   STATUS[293].TimeStamp := 16#0000;
   STATUS[294].EXT.AlarmWarnUnAck := FALSE;
   STATUS[294].EXT.AckRequired := FALSE;
   STATUS[294].EXT.Maintanence := FALSE;
   STATUS[294].EXT.Operation := FALSE;
   STATUS[294].EXT.Forced := FALSE;
   STATUS[294].EXT.BIT29 := FALSE;
   STATUS[294].EXT.BIT30 := FALSE;
   STATUS[294].EXT.BIT31 := FALSE;
   STATUS[294].EXT.ModeBit1 := FALSE;
   STATUS[294].EXT.ModeBit2 := FALSE;
   STATUS[294].EXT.ModeBit3 := FALSE;
   STATUS[294].EXT.BIT19 := FALSE;
   STATUS[294].EXT.BIT20 := FALSE;
   STATUS[294].EXT.AlarmSuppressed := FALSE;
   STATUS[294].EXT.AlarmPresent := FALSE;
   STATUS[294].EXT.AlarmFailUnAck := FALSE;
   STATUS[294].Status := 0;
   STATUS[294].TimeStamp := 16#0000;
   STATUS[295].EXT.AlarmWarnUnAck := FALSE;
   STATUS[295].EXT.AckRequired := FALSE;
   STATUS[295].EXT.Maintanence := FALSE;
   STATUS[295].EXT.Operation := FALSE;
   STATUS[295].EXT.Forced := FALSE;
   STATUS[295].EXT.BIT29 := FALSE;
   STATUS[295].EXT.BIT30 := FALSE;
   STATUS[295].EXT.BIT31 := FALSE;
   STATUS[295].EXT.ModeBit1 := FALSE;
   STATUS[295].EXT.ModeBit2 := FALSE;
   STATUS[295].EXT.ModeBit3 := FALSE;
   STATUS[295].EXT.BIT19 := FALSE;
   STATUS[295].EXT.BIT20 := FALSE;
   STATUS[295].EXT.AlarmSuppressed := FALSE;
   STATUS[295].EXT.AlarmPresent := FALSE;
   STATUS[295].EXT.AlarmFailUnAck := FALSE;
   STATUS[295].Status := 0;
   STATUS[295].TimeStamp := 16#0000;
   STATUS[296].EXT.AlarmWarnUnAck := FALSE;
   STATUS[296].EXT.AckRequired := FALSE;
   STATUS[296].EXT.Maintanence := FALSE;
   STATUS[296].EXT.Operation := FALSE;
   STATUS[296].EXT.Forced := FALSE;
   STATUS[296].EXT.BIT29 := FALSE;
   STATUS[296].EXT.BIT30 := FALSE;
   STATUS[296].EXT.BIT31 := FALSE;
   STATUS[296].EXT.ModeBit1 := FALSE;
   STATUS[296].EXT.ModeBit2 := FALSE;
   STATUS[296].EXT.ModeBit3 := FALSE;
   STATUS[296].EXT.BIT19 := FALSE;
   STATUS[296].EXT.BIT20 := FALSE;
   STATUS[296].EXT.AlarmSuppressed := FALSE;
   STATUS[296].EXT.AlarmPresent := FALSE;
   STATUS[296].EXT.AlarmFailUnAck := FALSE;
   STATUS[296].Status := 0;
   STATUS[296].TimeStamp := 16#0000;
   STATUS[297].EXT.AlarmWarnUnAck := FALSE;
   STATUS[297].EXT.AckRequired := FALSE;
   STATUS[297].EXT.Maintanence := FALSE;
   STATUS[297].EXT.Operation := FALSE;
   STATUS[297].EXT.Forced := FALSE;
   STATUS[297].EXT.BIT29 := FALSE;
   STATUS[297].EXT.BIT30 := FALSE;
   STATUS[297].EXT.BIT31 := FALSE;
   STATUS[297].EXT.ModeBit1 := FALSE;
   STATUS[297].EXT.ModeBit2 := FALSE;
   STATUS[297].EXT.ModeBit3 := FALSE;
   STATUS[297].EXT.BIT19 := FALSE;
   STATUS[297].EXT.BIT20 := FALSE;
   STATUS[297].EXT.AlarmSuppressed := FALSE;
   STATUS[297].EXT.AlarmPresent := FALSE;
   STATUS[297].EXT.AlarmFailUnAck := FALSE;
   STATUS[297].Status := 0;
   STATUS[297].TimeStamp := 16#0000;
   STATUS[298].EXT.AlarmWarnUnAck := FALSE;
   STATUS[298].EXT.AckRequired := FALSE;
   STATUS[298].EXT.Maintanence := FALSE;
   STATUS[298].EXT.Operation := FALSE;
   STATUS[298].EXT.Forced := FALSE;
   STATUS[298].EXT.BIT29 := FALSE;
   STATUS[298].EXT.BIT30 := FALSE;
   STATUS[298].EXT.BIT31 := FALSE;
   STATUS[298].EXT.ModeBit1 := FALSE;
   STATUS[298].EXT.ModeBit2 := FALSE;
   STATUS[298].EXT.ModeBit3 := FALSE;
   STATUS[298].EXT.BIT19 := FALSE;
   STATUS[298].EXT.BIT20 := FALSE;
   STATUS[298].EXT.AlarmSuppressed := FALSE;
   STATUS[298].EXT.AlarmPresent := FALSE;
   STATUS[298].EXT.AlarmFailUnAck := FALSE;
   STATUS[298].Status := 0;
   STATUS[298].TimeStamp := 16#0000;
   STATUS[299].EXT.AlarmWarnUnAck := FALSE;
   STATUS[299].EXT.AckRequired := FALSE;
   STATUS[299].EXT.Maintanence := FALSE;
   STATUS[299].EXT.Operation := FALSE;
   STATUS[299].EXT.Forced := FALSE;
   STATUS[299].EXT.BIT29 := FALSE;
   STATUS[299].EXT.BIT30 := FALSE;
   STATUS[299].EXT.BIT31 := FALSE;
   STATUS[299].EXT.ModeBit1 := FALSE;
   STATUS[299].EXT.ModeBit2 := FALSE;
   STATUS[299].EXT.ModeBit3 := FALSE;
   STATUS[299].EXT.BIT19 := FALSE;
   STATUS[299].EXT.BIT20 := FALSE;
   STATUS[299].EXT.AlarmSuppressed := FALSE;
   STATUS[299].EXT.AlarmPresent := FALSE;
   STATUS[299].EXT.AlarmFailUnAck := FALSE;
   STATUS[299].Status := 0;
   STATUS[299].TimeStamp := 16#0000;
   STATUS[300].EXT.AlarmWarnUnAck := FALSE;
   STATUS[300].EXT.AckRequired := FALSE;
   STATUS[300].EXT.Maintanence := FALSE;
   STATUS[300].EXT.Operation := FALSE;
   STATUS[300].EXT.Forced := FALSE;
   STATUS[300].EXT.BIT29 := FALSE;
   STATUS[300].EXT.BIT30 := FALSE;
   STATUS[300].EXT.BIT31 := FALSE;
   STATUS[300].EXT.ModeBit1 := FALSE;
   STATUS[300].EXT.ModeBit2 := FALSE;
   STATUS[300].EXT.ModeBit3 := FALSE;
   STATUS[300].EXT.BIT19 := FALSE;
   STATUS[300].EXT.BIT20 := FALSE;
   STATUS[300].EXT.AlarmSuppressed := FALSE;
   STATUS[300].EXT.AlarmPresent := FALSE;
   STATUS[300].EXT.AlarmFailUnAck := FALSE;
   STATUS[300].Status := 0;
   STATUS[300].TimeStamp := 16#0000;
   STATUS[301].EXT.AlarmWarnUnAck := FALSE;
   STATUS[301].EXT.AckRequired := FALSE;
   STATUS[301].EXT.Maintanence := FALSE;
   STATUS[301].EXT.Operation := FALSE;
   STATUS[301].EXT.Forced := FALSE;
   STATUS[301].EXT.BIT29 := FALSE;
   STATUS[301].EXT.BIT30 := FALSE;
   STATUS[301].EXT.BIT31 := FALSE;
   STATUS[301].EXT.ModeBit1 := FALSE;
   STATUS[301].EXT.ModeBit2 := FALSE;
   STATUS[301].EXT.ModeBit3 := FALSE;
   STATUS[301].EXT.BIT19 := FALSE;
   STATUS[301].EXT.BIT20 := FALSE;
   STATUS[301].EXT.AlarmSuppressed := FALSE;
   STATUS[301].EXT.AlarmPresent := FALSE;
   STATUS[301].EXT.AlarmFailUnAck := FALSE;
   STATUS[301].Status := 0;
   STATUS[301].TimeStamp := 16#0000;
   STATUS[302].EXT.AlarmWarnUnAck := FALSE;
   STATUS[302].EXT.AckRequired := FALSE;
   STATUS[302].EXT.Maintanence := FALSE;
   STATUS[302].EXT.Operation := FALSE;
   STATUS[302].EXT.Forced := FALSE;
   STATUS[302].EXT.BIT29 := FALSE;
   STATUS[302].EXT.BIT30 := FALSE;
   STATUS[302].EXT.BIT31 := FALSE;
   STATUS[302].EXT.ModeBit1 := FALSE;
   STATUS[302].EXT.ModeBit2 := FALSE;
   STATUS[302].EXT.ModeBit3 := FALSE;
   STATUS[302].EXT.BIT19 := FALSE;
   STATUS[302].EXT.BIT20 := FALSE;
   STATUS[302].EXT.AlarmSuppressed := FALSE;
   STATUS[302].EXT.AlarmPresent := FALSE;
   STATUS[302].EXT.AlarmFailUnAck := FALSE;
   STATUS[302].Status := 0;
   STATUS[302].TimeStamp := 16#0000;
   STATUS[303].EXT.AlarmWarnUnAck := FALSE;
   STATUS[303].EXT.AckRequired := FALSE;
   STATUS[303].EXT.Maintanence := FALSE;
   STATUS[303].EXT.Operation := FALSE;
   STATUS[303].EXT.Forced := FALSE;
   STATUS[303].EXT.BIT29 := FALSE;
   STATUS[303].EXT.BIT30 := FALSE;
   STATUS[303].EXT.BIT31 := FALSE;
   STATUS[303].EXT.ModeBit1 := FALSE;
   STATUS[303].EXT.ModeBit2 := FALSE;
   STATUS[303].EXT.ModeBit3 := FALSE;
   STATUS[303].EXT.BIT19 := FALSE;
   STATUS[303].EXT.BIT20 := FALSE;
   STATUS[303].EXT.AlarmSuppressed := FALSE;
   STATUS[303].EXT.AlarmPresent := FALSE;
   STATUS[303].EXT.AlarmFailUnAck := FALSE;
   STATUS[303].Status := 0;
   STATUS[303].TimeStamp := 16#0000;
   STATUS[304].EXT.AlarmWarnUnAck := FALSE;
   STATUS[304].EXT.AckRequired := FALSE;
   STATUS[304].EXT.Maintanence := FALSE;
   STATUS[304].EXT.Operation := FALSE;
   STATUS[304].EXT.Forced := FALSE;
   STATUS[304].EXT.BIT29 := FALSE;
   STATUS[304].EXT.BIT30 := FALSE;
   STATUS[304].EXT.BIT31 := FALSE;
   STATUS[304].EXT.ModeBit1 := FALSE;
   STATUS[304].EXT.ModeBit2 := FALSE;
   STATUS[304].EXT.ModeBit3 := FALSE;
   STATUS[304].EXT.BIT19 := FALSE;
   STATUS[304].EXT.BIT20 := FALSE;
   STATUS[304].EXT.AlarmSuppressed := FALSE;
   STATUS[304].EXT.AlarmPresent := FALSE;
   STATUS[304].EXT.AlarmFailUnAck := FALSE;
   STATUS[304].Status := 0;
   STATUS[304].TimeStamp := 16#0000;
   STATUS[305].EXT.AlarmWarnUnAck := FALSE;
   STATUS[305].EXT.AckRequired := FALSE;
   STATUS[305].EXT.Maintanence := FALSE;
   STATUS[305].EXT.Operation := FALSE;
   STATUS[305].EXT.Forced := FALSE;
   STATUS[305].EXT.BIT29 := FALSE;
   STATUS[305].EXT.BIT30 := FALSE;
   STATUS[305].EXT.BIT31 := FALSE;
   STATUS[305].EXT.ModeBit1 := FALSE;
   STATUS[305].EXT.ModeBit2 := FALSE;
   STATUS[305].EXT.ModeBit3 := FALSE;
   STATUS[305].EXT.BIT19 := FALSE;
   STATUS[305].EXT.BIT20 := FALSE;
   STATUS[305].EXT.AlarmSuppressed := FALSE;
   STATUS[305].EXT.AlarmPresent := FALSE;
   STATUS[305].EXT.AlarmFailUnAck := FALSE;
   STATUS[305].Status := 0;
   STATUS[305].TimeStamp := 16#0000;
   STATUS[306].EXT.AlarmWarnUnAck := FALSE;
   STATUS[306].EXT.AckRequired := FALSE;
   STATUS[306].EXT.Maintanence := FALSE;
   STATUS[306].EXT.Operation := FALSE;
   STATUS[306].EXT.Forced := FALSE;
   STATUS[306].EXT.BIT29 := FALSE;
   STATUS[306].EXT.BIT30 := FALSE;
   STATUS[306].EXT.BIT31 := FALSE;
   STATUS[306].EXT.ModeBit1 := FALSE;
   STATUS[306].EXT.ModeBit2 := FALSE;
   STATUS[306].EXT.ModeBit3 := FALSE;
   STATUS[306].EXT.BIT19 := FALSE;
   STATUS[306].EXT.BIT20 := FALSE;
   STATUS[306].EXT.AlarmSuppressed := FALSE;
   STATUS[306].EXT.AlarmPresent := FALSE;
   STATUS[306].EXT.AlarmFailUnAck := FALSE;
   STATUS[306].Status := 0;
   STATUS[306].TimeStamp := 16#0000;
   STATUS[307].EXT.AlarmWarnUnAck := FALSE;
   STATUS[307].EXT.AckRequired := FALSE;
   STATUS[307].EXT.Maintanence := FALSE;
   STATUS[307].EXT.Operation := FALSE;
   STATUS[307].EXT.Forced := FALSE;
   STATUS[307].EXT.BIT29 := FALSE;
   STATUS[307].EXT.BIT30 := FALSE;
   STATUS[307].EXT.BIT31 := FALSE;
   STATUS[307].EXT.ModeBit1 := FALSE;
   STATUS[307].EXT.ModeBit2 := FALSE;
   STATUS[307].EXT.ModeBit3 := FALSE;
   STATUS[307].EXT.BIT19 := FALSE;
   STATUS[307].EXT.BIT20 := FALSE;
   STATUS[307].EXT.AlarmSuppressed := FALSE;
   STATUS[307].EXT.AlarmPresent := FALSE;
   STATUS[307].EXT.AlarmFailUnAck := FALSE;
   STATUS[307].Status := 0;
   STATUS[307].TimeStamp := 16#0000;
   STATUS[308].EXT.AlarmWarnUnAck := FALSE;
   STATUS[308].EXT.AckRequired := FALSE;
   STATUS[308].EXT.Maintanence := FALSE;
   STATUS[308].EXT.Operation := FALSE;
   STATUS[308].EXT.Forced := FALSE;
   STATUS[308].EXT.BIT29 := FALSE;
   STATUS[308].EXT.BIT30 := FALSE;
   STATUS[308].EXT.BIT31 := FALSE;
   STATUS[308].EXT.ModeBit1 := FALSE;
   STATUS[308].EXT.ModeBit2 := FALSE;
   STATUS[308].EXT.ModeBit3 := FALSE;
   STATUS[308].EXT.BIT19 := FALSE;
   STATUS[308].EXT.BIT20 := FALSE;
   STATUS[308].EXT.AlarmSuppressed := FALSE;
   STATUS[308].EXT.AlarmPresent := FALSE;
   STATUS[308].EXT.AlarmFailUnAck := FALSE;
   STATUS[308].Status := 0;
   STATUS[308].TimeStamp := 16#0000;
   STATUS[309].EXT.AlarmWarnUnAck := FALSE;
   STATUS[309].EXT.AckRequired := FALSE;
   STATUS[309].EXT.Maintanence := FALSE;
   STATUS[309].EXT.Operation := FALSE;
   STATUS[309].EXT.Forced := FALSE;
   STATUS[309].EXT.BIT29 := FALSE;
   STATUS[309].EXT.BIT30 := FALSE;
   STATUS[309].EXT.BIT31 := FALSE;
   STATUS[309].EXT.ModeBit1 := FALSE;
   STATUS[309].EXT.ModeBit2 := FALSE;
   STATUS[309].EXT.ModeBit3 := FALSE;
   STATUS[309].EXT.BIT19 := FALSE;
   STATUS[309].EXT.BIT20 := FALSE;
   STATUS[309].EXT.AlarmSuppressed := FALSE;
   STATUS[309].EXT.AlarmPresent := FALSE;
   STATUS[309].EXT.AlarmFailUnAck := FALSE;
   STATUS[309].Status := 0;
   STATUS[309].TimeStamp := 16#0000;
   STATUS[310].EXT.AlarmWarnUnAck := FALSE;
   STATUS[310].EXT.AckRequired := FALSE;
   STATUS[310].EXT.Maintanence := FALSE;
   STATUS[310].EXT.Operation := FALSE;
   STATUS[310].EXT.Forced := FALSE;
   STATUS[310].EXT.BIT29 := FALSE;
   STATUS[310].EXT.BIT30 := FALSE;
   STATUS[310].EXT.BIT31 := FALSE;
   STATUS[310].EXT.ModeBit1 := FALSE;
   STATUS[310].EXT.ModeBit2 := FALSE;
   STATUS[310].EXT.ModeBit3 := FALSE;
   STATUS[310].EXT.BIT19 := FALSE;
   STATUS[310].EXT.BIT20 := FALSE;
   STATUS[310].EXT.AlarmSuppressed := FALSE;
   STATUS[310].EXT.AlarmPresent := FALSE;
   STATUS[310].EXT.AlarmFailUnAck := FALSE;
   STATUS[310].Status := 0;
   STATUS[310].TimeStamp := 16#0000;
   STATUS[311].EXT.AlarmWarnUnAck := FALSE;
   STATUS[311].EXT.AckRequired := FALSE;
   STATUS[311].EXT.Maintanence := FALSE;
   STATUS[311].EXT.Operation := FALSE;
   STATUS[311].EXT.Forced := FALSE;
   STATUS[311].EXT.BIT29 := FALSE;
   STATUS[311].EXT.BIT30 := FALSE;
   STATUS[311].EXT.BIT31 := FALSE;
   STATUS[311].EXT.ModeBit1 := FALSE;
   STATUS[311].EXT.ModeBit2 := FALSE;
   STATUS[311].EXT.ModeBit3 := FALSE;
   STATUS[311].EXT.BIT19 := FALSE;
   STATUS[311].EXT.BIT20 := FALSE;
   STATUS[311].EXT.AlarmSuppressed := FALSE;
   STATUS[311].EXT.AlarmPresent := FALSE;
   STATUS[311].EXT.AlarmFailUnAck := FALSE;
   STATUS[311].Status := 0;
   STATUS[311].TimeStamp := 16#0000;
   STATUS[312].EXT.AlarmWarnUnAck := FALSE;
   STATUS[312].EXT.AckRequired := FALSE;
   STATUS[312].EXT.Maintanence := FALSE;
   STATUS[312].EXT.Operation := FALSE;
   STATUS[312].EXT.Forced := FALSE;
   STATUS[312].EXT.BIT29 := FALSE;
   STATUS[312].EXT.BIT30 := FALSE;
   STATUS[312].EXT.BIT31 := FALSE;
   STATUS[312].EXT.ModeBit1 := FALSE;
   STATUS[312].EXT.ModeBit2 := FALSE;
   STATUS[312].EXT.ModeBit3 := FALSE;
   STATUS[312].EXT.BIT19 := FALSE;
   STATUS[312].EXT.BIT20 := FALSE;
   STATUS[312].EXT.AlarmSuppressed := FALSE;
   STATUS[312].EXT.AlarmPresent := FALSE;
   STATUS[312].EXT.AlarmFailUnAck := FALSE;
   STATUS[312].Status := 0;
   STATUS[312].TimeStamp := 16#0000;
   STATUS[313].EXT.AlarmWarnUnAck := FALSE;
   STATUS[313].EXT.AckRequired := FALSE;
   STATUS[313].EXT.Maintanence := FALSE;
   STATUS[313].EXT.Operation := FALSE;
   STATUS[313].EXT.Forced := FALSE;
   STATUS[313].EXT.BIT29 := FALSE;
   STATUS[313].EXT.BIT30 := FALSE;
   STATUS[313].EXT.BIT31 := FALSE;
   STATUS[313].EXT.ModeBit1 := FALSE;
   STATUS[313].EXT.ModeBit2 := FALSE;
   STATUS[313].EXT.ModeBit3 := FALSE;
   STATUS[313].EXT.BIT19 := FALSE;
   STATUS[313].EXT.BIT20 := FALSE;
   STATUS[313].EXT.AlarmSuppressed := FALSE;
   STATUS[313].EXT.AlarmPresent := FALSE;
   STATUS[313].EXT.AlarmFailUnAck := FALSE;
   STATUS[313].Status := 0;
   STATUS[313].TimeStamp := 16#0000;
   STATUS[314].EXT.AlarmWarnUnAck := FALSE;
   STATUS[314].EXT.AckRequired := FALSE;
   STATUS[314].EXT.Maintanence := FALSE;
   STATUS[314].EXT.Operation := FALSE;
   STATUS[314].EXT.Forced := FALSE;
   STATUS[314].EXT.BIT29 := FALSE;
   STATUS[314].EXT.BIT30 := FALSE;
   STATUS[314].EXT.BIT31 := FALSE;
   STATUS[314].EXT.ModeBit1 := FALSE;
   STATUS[314].EXT.ModeBit2 := FALSE;
   STATUS[314].EXT.ModeBit3 := FALSE;
   STATUS[314].EXT.BIT19 := FALSE;
   STATUS[314].EXT.BIT20 := FALSE;
   STATUS[314].EXT.AlarmSuppressed := FALSE;
   STATUS[314].EXT.AlarmPresent := FALSE;
   STATUS[314].EXT.AlarmFailUnAck := FALSE;
   STATUS[314].Status := 0;
   STATUS[314].TimeStamp := 16#0000;
   STATUS[315].EXT.AlarmWarnUnAck := FALSE;
   STATUS[315].EXT.AckRequired := FALSE;
   STATUS[315].EXT.Maintanence := FALSE;
   STATUS[315].EXT.Operation := FALSE;
   STATUS[315].EXT.Forced := FALSE;
   STATUS[315].EXT.BIT29 := FALSE;
   STATUS[315].EXT.BIT30 := FALSE;
   STATUS[315].EXT.BIT31 := FALSE;
   STATUS[315].EXT.ModeBit1 := FALSE;
   STATUS[315].EXT.ModeBit2 := FALSE;
   STATUS[315].EXT.ModeBit3 := FALSE;
   STATUS[315].EXT.BIT19 := FALSE;
   STATUS[315].EXT.BIT20 := FALSE;
   STATUS[315].EXT.AlarmSuppressed := FALSE;
   STATUS[315].EXT.AlarmPresent := FALSE;
   STATUS[315].EXT.AlarmFailUnAck := FALSE;
   STATUS[315].Status := 0;
   STATUS[315].TimeStamp := 16#0000;
   STATUS[316].EXT.AlarmWarnUnAck := FALSE;
   STATUS[316].EXT.AckRequired := FALSE;
   STATUS[316].EXT.Maintanence := FALSE;
   STATUS[316].EXT.Operation := FALSE;
   STATUS[316].EXT.Forced := FALSE;
   STATUS[316].EXT.BIT29 := FALSE;
   STATUS[316].EXT.BIT30 := FALSE;
   STATUS[316].EXT.BIT31 := FALSE;
   STATUS[316].EXT.ModeBit1 := FALSE;
   STATUS[316].EXT.ModeBit2 := FALSE;
   STATUS[316].EXT.ModeBit3 := FALSE;
   STATUS[316].EXT.BIT19 := FALSE;
   STATUS[316].EXT.BIT20 := FALSE;
   STATUS[316].EXT.AlarmSuppressed := FALSE;
   STATUS[316].EXT.AlarmPresent := FALSE;
   STATUS[316].EXT.AlarmFailUnAck := FALSE;
   STATUS[316].Status := 0;
   STATUS[316].TimeStamp := 16#0000;
   STATUS[317].EXT.AlarmWarnUnAck := FALSE;
   STATUS[317].EXT.AckRequired := FALSE;
   STATUS[317].EXT.Maintanence := FALSE;
   STATUS[317].EXT.Operation := FALSE;
   STATUS[317].EXT.Forced := FALSE;
   STATUS[317].EXT.BIT29 := FALSE;
   STATUS[317].EXT.BIT30 := FALSE;
   STATUS[317].EXT.BIT31 := FALSE;
   STATUS[317].EXT.ModeBit1 := FALSE;
   STATUS[317].EXT.ModeBit2 := FALSE;
   STATUS[317].EXT.ModeBit3 := FALSE;
   STATUS[317].EXT.BIT19 := FALSE;
   STATUS[317].EXT.BIT20 := FALSE;
   STATUS[317].EXT.AlarmSuppressed := FALSE;
   STATUS[317].EXT.AlarmPresent := FALSE;
   STATUS[317].EXT.AlarmFailUnAck := FALSE;
   STATUS[317].Status := 0;
   STATUS[317].TimeStamp := 16#0000;
   STATUS[318].EXT.AlarmWarnUnAck := FALSE;
   STATUS[318].EXT.AckRequired := FALSE;
   STATUS[318].EXT.Maintanence := FALSE;
   STATUS[318].EXT.Operation := FALSE;
   STATUS[318].EXT.Forced := FALSE;
   STATUS[318].EXT.BIT29 := FALSE;
   STATUS[318].EXT.BIT30 := FALSE;
   STATUS[318].EXT.BIT31 := FALSE;
   STATUS[318].EXT.ModeBit1 := FALSE;
   STATUS[318].EXT.ModeBit2 := FALSE;
   STATUS[318].EXT.ModeBit3 := FALSE;
   STATUS[318].EXT.BIT19 := FALSE;
   STATUS[318].EXT.BIT20 := FALSE;
   STATUS[318].EXT.AlarmSuppressed := FALSE;
   STATUS[318].EXT.AlarmPresent := FALSE;
   STATUS[318].EXT.AlarmFailUnAck := FALSE;
   STATUS[318].Status := 0;
   STATUS[318].TimeStamp := 16#0000;
   STATUS[319].EXT.AlarmWarnUnAck := FALSE;
   STATUS[319].EXT.AckRequired := FALSE;
   STATUS[319].EXT.Maintanence := FALSE;
   STATUS[319].EXT.Operation := FALSE;
   STATUS[319].EXT.Forced := FALSE;
   STATUS[319].EXT.BIT29 := FALSE;
   STATUS[319].EXT.BIT30 := FALSE;
   STATUS[319].EXT.BIT31 := FALSE;
   STATUS[319].EXT.ModeBit1 := FALSE;
   STATUS[319].EXT.ModeBit2 := FALSE;
   STATUS[319].EXT.ModeBit3 := FALSE;
   STATUS[319].EXT.BIT19 := FALSE;
   STATUS[319].EXT.BIT20 := FALSE;
   STATUS[319].EXT.AlarmSuppressed := FALSE;
   STATUS[319].EXT.AlarmPresent := FALSE;
   STATUS[319].EXT.AlarmFailUnAck := FALSE;
   STATUS[319].Status := 0;
   STATUS[319].TimeStamp := 16#0000;
   STATUS[320].EXT.AlarmWarnUnAck := FALSE;
   STATUS[320].EXT.AckRequired := FALSE;
   STATUS[320].EXT.Maintanence := FALSE;
   STATUS[320].EXT.Operation := FALSE;
   STATUS[320].EXT.Forced := FALSE;
   STATUS[320].EXT.BIT29 := FALSE;
   STATUS[320].EXT.BIT30 := FALSE;
   STATUS[320].EXT.BIT31 := FALSE;
   STATUS[320].EXT.ModeBit1 := FALSE;
   STATUS[320].EXT.ModeBit2 := FALSE;
   STATUS[320].EXT.ModeBit3 := FALSE;
   STATUS[320].EXT.BIT19 := FALSE;
   STATUS[320].EXT.BIT20 := FALSE;
   STATUS[320].EXT.AlarmSuppressed := FALSE;
   STATUS[320].EXT.AlarmPresent := FALSE;
   STATUS[320].EXT.AlarmFailUnAck := FALSE;
   STATUS[320].Status := 0;
   STATUS[320].TimeStamp := 16#0000;
   STATUS[321].EXT.AlarmWarnUnAck := FALSE;
   STATUS[321].EXT.AckRequired := FALSE;
   STATUS[321].EXT.Maintanence := FALSE;
   STATUS[321].EXT.Operation := FALSE;
   STATUS[321].EXT.Forced := FALSE;
   STATUS[321].EXT.BIT29 := FALSE;
   STATUS[321].EXT.BIT30 := FALSE;
   STATUS[321].EXT.BIT31 := FALSE;
   STATUS[321].EXT.ModeBit1 := FALSE;
   STATUS[321].EXT.ModeBit2 := FALSE;
   STATUS[321].EXT.ModeBit3 := FALSE;
   STATUS[321].EXT.BIT19 := FALSE;
   STATUS[321].EXT.BIT20 := FALSE;
   STATUS[321].EXT.AlarmSuppressed := FALSE;
   STATUS[321].EXT.AlarmPresent := FALSE;
   STATUS[321].EXT.AlarmFailUnAck := FALSE;
   STATUS[321].Status := 0;
   STATUS[321].TimeStamp := 16#0000;
   STATUS[322].EXT.AlarmWarnUnAck := FALSE;
   STATUS[322].EXT.AckRequired := FALSE;
   STATUS[322].EXT.Maintanence := FALSE;
   STATUS[322].EXT.Operation := FALSE;
   STATUS[322].EXT.Forced := FALSE;
   STATUS[322].EXT.BIT29 := FALSE;
   STATUS[322].EXT.BIT30 := FALSE;
   STATUS[322].EXT.BIT31 := FALSE;
   STATUS[322].EXT.ModeBit1 := FALSE;
   STATUS[322].EXT.ModeBit2 := FALSE;
   STATUS[322].EXT.ModeBit3 := FALSE;
   STATUS[322].EXT.BIT19 := FALSE;
   STATUS[322].EXT.BIT20 := FALSE;
   STATUS[322].EXT.AlarmSuppressed := FALSE;
   STATUS[322].EXT.AlarmPresent := FALSE;
   STATUS[322].EXT.AlarmFailUnAck := FALSE;
   STATUS[322].Status := 0;
   STATUS[322].TimeStamp := 16#0000;
   STATUS[323].EXT.AlarmWarnUnAck := FALSE;
   STATUS[323].EXT.AckRequired := FALSE;
   STATUS[323].EXT.Maintanence := FALSE;
   STATUS[323].EXT.Operation := FALSE;
   STATUS[323].EXT.Forced := FALSE;
   STATUS[323].EXT.BIT29 := FALSE;
   STATUS[323].EXT.BIT30 := FALSE;
   STATUS[323].EXT.BIT31 := FALSE;
   STATUS[323].EXT.ModeBit1 := FALSE;
   STATUS[323].EXT.ModeBit2 := FALSE;
   STATUS[323].EXT.ModeBit3 := FALSE;
   STATUS[323].EXT.BIT19 := FALSE;
   STATUS[323].EXT.BIT20 := FALSE;
   STATUS[323].EXT.AlarmSuppressed := FALSE;
   STATUS[323].EXT.AlarmPresent := FALSE;
   STATUS[323].EXT.AlarmFailUnAck := FALSE;
   STATUS[323].Status := 0;
   STATUS[323].TimeStamp := 16#0000;
   STATUS[324].EXT.AlarmWarnUnAck := FALSE;
   STATUS[324].EXT.AckRequired := FALSE;
   STATUS[324].EXT.Maintanence := FALSE;
   STATUS[324].EXT.Operation := FALSE;
   STATUS[324].EXT.Forced := FALSE;
   STATUS[324].EXT.BIT29 := FALSE;
   STATUS[324].EXT.BIT30 := FALSE;
   STATUS[324].EXT.BIT31 := FALSE;
   STATUS[324].EXT.ModeBit1 := FALSE;
   STATUS[324].EXT.ModeBit2 := FALSE;
   STATUS[324].EXT.ModeBit3 := FALSE;
   STATUS[324].EXT.BIT19 := FALSE;
   STATUS[324].EXT.BIT20 := FALSE;
   STATUS[324].EXT.AlarmSuppressed := FALSE;
   STATUS[324].EXT.AlarmPresent := FALSE;
   STATUS[324].EXT.AlarmFailUnAck := FALSE;
   STATUS[324].Status := 0;
   STATUS[324].TimeStamp := 16#0000;
   STATUS[325].EXT.AlarmWarnUnAck := FALSE;
   STATUS[325].EXT.AckRequired := FALSE;
   STATUS[325].EXT.Maintanence := FALSE;
   STATUS[325].EXT.Operation := FALSE;
   STATUS[325].EXT.Forced := FALSE;
   STATUS[325].EXT.BIT29 := FALSE;
   STATUS[325].EXT.BIT30 := FALSE;
   STATUS[325].EXT.BIT31 := FALSE;
   STATUS[325].EXT.ModeBit1 := FALSE;
   STATUS[325].EXT.ModeBit2 := FALSE;
   STATUS[325].EXT.ModeBit3 := FALSE;
   STATUS[325].EXT.BIT19 := FALSE;
   STATUS[325].EXT.BIT20 := FALSE;
   STATUS[325].EXT.AlarmSuppressed := FALSE;
   STATUS[325].EXT.AlarmPresent := FALSE;
   STATUS[325].EXT.AlarmFailUnAck := FALSE;
   STATUS[325].Status := 0;
   STATUS[325].TimeStamp := 16#0000;
   STATUS[326].EXT.AlarmWarnUnAck := FALSE;
   STATUS[326].EXT.AckRequired := FALSE;
   STATUS[326].EXT.Maintanence := FALSE;
   STATUS[326].EXT.Operation := FALSE;
   STATUS[326].EXT.Forced := FALSE;
   STATUS[326].EXT.BIT29 := FALSE;
   STATUS[326].EXT.BIT30 := FALSE;
   STATUS[326].EXT.BIT31 := FALSE;
   STATUS[326].EXT.ModeBit1 := FALSE;
   STATUS[326].EXT.ModeBit2 := FALSE;
   STATUS[326].EXT.ModeBit3 := FALSE;
   STATUS[326].EXT.BIT19 := FALSE;
   STATUS[326].EXT.BIT20 := FALSE;
   STATUS[326].EXT.AlarmSuppressed := FALSE;
   STATUS[326].EXT.AlarmPresent := FALSE;
   STATUS[326].EXT.AlarmFailUnAck := FALSE;
   STATUS[326].Status := 0;
   STATUS[326].TimeStamp := 16#0000;
   STATUS[327].EXT.AlarmWarnUnAck := FALSE;
   STATUS[327].EXT.AckRequired := FALSE;
   STATUS[327].EXT.Maintanence := FALSE;
   STATUS[327].EXT.Operation := FALSE;
   STATUS[327].EXT.Forced := FALSE;
   STATUS[327].EXT.BIT29 := FALSE;
   STATUS[327].EXT.BIT30 := FALSE;
   STATUS[327].EXT.BIT31 := FALSE;
   STATUS[327].EXT.ModeBit1 := FALSE;
   STATUS[327].EXT.ModeBit2 := FALSE;
   STATUS[327].EXT.ModeBit3 := FALSE;
   STATUS[327].EXT.BIT19 := FALSE;
   STATUS[327].EXT.BIT20 := FALSE;
   STATUS[327].EXT.AlarmSuppressed := FALSE;
   STATUS[327].EXT.AlarmPresent := FALSE;
   STATUS[327].EXT.AlarmFailUnAck := FALSE;
   STATUS[327].Status := 0;
   STATUS[327].TimeStamp := 16#0000;
   STATUS[328].EXT.AlarmWarnUnAck := FALSE;
   STATUS[328].EXT.AckRequired := FALSE;
   STATUS[328].EXT.Maintanence := FALSE;
   STATUS[328].EXT.Operation := FALSE;
   STATUS[328].EXT.Forced := FALSE;
   STATUS[328].EXT.BIT29 := FALSE;
   STATUS[328].EXT.BIT30 := FALSE;
   STATUS[328].EXT.BIT31 := FALSE;
   STATUS[328].EXT.ModeBit1 := FALSE;
   STATUS[328].EXT.ModeBit2 := FALSE;
   STATUS[328].EXT.ModeBit3 := FALSE;
   STATUS[328].EXT.BIT19 := FALSE;
   STATUS[328].EXT.BIT20 := FALSE;
   STATUS[328].EXT.AlarmSuppressed := FALSE;
   STATUS[328].EXT.AlarmPresent := FALSE;
   STATUS[328].EXT.AlarmFailUnAck := FALSE;
   STATUS[328].Status := 0;
   STATUS[328].TimeStamp := 16#0000;
   STATUS[329].EXT.AlarmWarnUnAck := FALSE;
   STATUS[329].EXT.AckRequired := FALSE;
   STATUS[329].EXT.Maintanence := FALSE;
   STATUS[329].EXT.Operation := FALSE;
   STATUS[329].EXT.Forced := FALSE;
   STATUS[329].EXT.BIT29 := FALSE;
   STATUS[329].EXT.BIT30 := FALSE;
   STATUS[329].EXT.BIT31 := FALSE;
   STATUS[329].EXT.ModeBit1 := FALSE;
   STATUS[329].EXT.ModeBit2 := FALSE;
   STATUS[329].EXT.ModeBit3 := FALSE;
   STATUS[329].EXT.BIT19 := FALSE;
   STATUS[329].EXT.BIT20 := FALSE;
   STATUS[329].EXT.AlarmSuppressed := FALSE;
   STATUS[329].EXT.AlarmPresent := FALSE;
   STATUS[329].EXT.AlarmFailUnAck := FALSE;
   STATUS[329].Status := 0;
   STATUS[329].TimeStamp := 16#0000;
   STATUS[330].EXT.AlarmWarnUnAck := FALSE;
   STATUS[330].EXT.AckRequired := FALSE;
   STATUS[330].EXT.Maintanence := FALSE;
   STATUS[330].EXT.Operation := FALSE;
   STATUS[330].EXT.Forced := FALSE;
   STATUS[330].EXT.BIT29 := FALSE;
   STATUS[330].EXT.BIT30 := FALSE;
   STATUS[330].EXT.BIT31 := FALSE;
   STATUS[330].EXT.ModeBit1 := FALSE;
   STATUS[330].EXT.ModeBit2 := FALSE;
   STATUS[330].EXT.ModeBit3 := FALSE;
   STATUS[330].EXT.BIT19 := FALSE;
   STATUS[330].EXT.BIT20 := FALSE;
   STATUS[330].EXT.AlarmSuppressed := FALSE;
   STATUS[330].EXT.AlarmPresent := FALSE;
   STATUS[330].EXT.AlarmFailUnAck := FALSE;
   STATUS[330].Status := 0;
   STATUS[330].TimeStamp := 16#0000;
   STATUS[331].EXT.AlarmWarnUnAck := FALSE;
   STATUS[331].EXT.AckRequired := FALSE;
   STATUS[331].EXT.Maintanence := FALSE;
   STATUS[331].EXT.Operation := FALSE;
   STATUS[331].EXT.Forced := FALSE;
   STATUS[331].EXT.BIT29 := FALSE;
   STATUS[331].EXT.BIT30 := FALSE;
   STATUS[331].EXT.BIT31 := FALSE;
   STATUS[331].EXT.ModeBit1 := FALSE;
   STATUS[331].EXT.ModeBit2 := FALSE;
   STATUS[331].EXT.ModeBit3 := FALSE;
   STATUS[331].EXT.BIT19 := FALSE;
   STATUS[331].EXT.BIT20 := FALSE;
   STATUS[331].EXT.AlarmSuppressed := FALSE;
   STATUS[331].EXT.AlarmPresent := FALSE;
   STATUS[331].EXT.AlarmFailUnAck := FALSE;
   STATUS[331].Status := 0;
   STATUS[331].TimeStamp := 16#0000;
   STATUS[332].EXT.AlarmWarnUnAck := FALSE;
   STATUS[332].EXT.AckRequired := FALSE;
   STATUS[332].EXT.Maintanence := FALSE;
   STATUS[332].EXT.Operation := FALSE;
   STATUS[332].EXT.Forced := FALSE;
   STATUS[332].EXT.BIT29 := FALSE;
   STATUS[332].EXT.BIT30 := FALSE;
   STATUS[332].EXT.BIT31 := FALSE;
   STATUS[332].EXT.ModeBit1 := FALSE;
   STATUS[332].EXT.ModeBit2 := FALSE;
   STATUS[332].EXT.ModeBit3 := FALSE;
   STATUS[332].EXT.BIT19 := FALSE;
   STATUS[332].EXT.BIT20 := FALSE;
   STATUS[332].EXT.AlarmSuppressed := FALSE;
   STATUS[332].EXT.AlarmPresent := FALSE;
   STATUS[332].EXT.AlarmFailUnAck := FALSE;
   STATUS[332].Status := 0;
   STATUS[332].TimeStamp := 16#0000;
   STATUS[333].EXT.AlarmWarnUnAck := FALSE;
   STATUS[333].EXT.AckRequired := FALSE;
   STATUS[333].EXT.Maintanence := FALSE;
   STATUS[333].EXT.Operation := FALSE;
   STATUS[333].EXT.Forced := FALSE;
   STATUS[333].EXT.BIT29 := FALSE;
   STATUS[333].EXT.BIT30 := FALSE;
   STATUS[333].EXT.BIT31 := FALSE;
   STATUS[333].EXT.ModeBit1 := FALSE;
   STATUS[333].EXT.ModeBit2 := FALSE;
   STATUS[333].EXT.ModeBit3 := FALSE;
   STATUS[333].EXT.BIT19 := FALSE;
   STATUS[333].EXT.BIT20 := FALSE;
   STATUS[333].EXT.AlarmSuppressed := FALSE;
   STATUS[333].EXT.AlarmPresent := FALSE;
   STATUS[333].EXT.AlarmFailUnAck := FALSE;
   STATUS[333].Status := 0;
   STATUS[333].TimeStamp := 16#0000;
   STATUS[334].EXT.AlarmWarnUnAck := FALSE;
   STATUS[334].EXT.AckRequired := FALSE;
   STATUS[334].EXT.Maintanence := FALSE;
   STATUS[334].EXT.Operation := FALSE;
   STATUS[334].EXT.Forced := FALSE;
   STATUS[334].EXT.BIT29 := FALSE;
   STATUS[334].EXT.BIT30 := FALSE;
   STATUS[334].EXT.BIT31 := FALSE;
   STATUS[334].EXT.ModeBit1 := FALSE;
   STATUS[334].EXT.ModeBit2 := FALSE;
   STATUS[334].EXT.ModeBit3 := FALSE;
   STATUS[334].EXT.BIT19 := FALSE;
   STATUS[334].EXT.BIT20 := FALSE;
   STATUS[334].EXT.AlarmSuppressed := FALSE;
   STATUS[334].EXT.AlarmPresent := FALSE;
   STATUS[334].EXT.AlarmFailUnAck := FALSE;
   STATUS[334].Status := 0;
   STATUS[334].TimeStamp := 16#0000;
   STATUS[335].EXT.AlarmWarnUnAck := FALSE;
   STATUS[335].EXT.AckRequired := FALSE;
   STATUS[335].EXT.Maintanence := FALSE;
   STATUS[335].EXT.Operation := FALSE;
   STATUS[335].EXT.Forced := FALSE;
   STATUS[335].EXT.BIT29 := FALSE;
   STATUS[335].EXT.BIT30 := FALSE;
   STATUS[335].EXT.BIT31 := FALSE;
   STATUS[335].EXT.ModeBit1 := FALSE;
   STATUS[335].EXT.ModeBit2 := FALSE;
   STATUS[335].EXT.ModeBit3 := FALSE;
   STATUS[335].EXT.BIT19 := FALSE;
   STATUS[335].EXT.BIT20 := FALSE;
   STATUS[335].EXT.AlarmSuppressed := FALSE;
   STATUS[335].EXT.AlarmPresent := FALSE;
   STATUS[335].EXT.AlarmFailUnAck := FALSE;
   STATUS[335].Status := 0;
   STATUS[335].TimeStamp := 16#0000;
   STATUS[336].EXT.AlarmWarnUnAck := FALSE;
   STATUS[336].EXT.AckRequired := FALSE;
   STATUS[336].EXT.Maintanence := FALSE;
   STATUS[336].EXT.Operation := FALSE;
   STATUS[336].EXT.Forced := FALSE;
   STATUS[336].EXT.BIT29 := FALSE;
   STATUS[336].EXT.BIT30 := FALSE;
   STATUS[336].EXT.BIT31 := FALSE;
   STATUS[336].EXT.ModeBit1 := FALSE;
   STATUS[336].EXT.ModeBit2 := FALSE;
   STATUS[336].EXT.ModeBit3 := FALSE;
   STATUS[336].EXT.BIT19 := FALSE;
   STATUS[336].EXT.BIT20 := FALSE;
   STATUS[336].EXT.AlarmSuppressed := FALSE;
   STATUS[336].EXT.AlarmPresent := FALSE;
   STATUS[336].EXT.AlarmFailUnAck := FALSE;
   STATUS[336].Status := 0;
   STATUS[336].TimeStamp := 16#0000;
   STATUS[337].EXT.AlarmWarnUnAck := FALSE;
   STATUS[337].EXT.AckRequired := FALSE;
   STATUS[337].EXT.Maintanence := FALSE;
   STATUS[337].EXT.Operation := FALSE;
   STATUS[337].EXT.Forced := FALSE;
   STATUS[337].EXT.BIT29 := FALSE;
   STATUS[337].EXT.BIT30 := FALSE;
   STATUS[337].EXT.BIT31 := FALSE;
   STATUS[337].EXT.ModeBit1 := FALSE;
   STATUS[337].EXT.ModeBit2 := FALSE;
   STATUS[337].EXT.ModeBit3 := FALSE;
   STATUS[337].EXT.BIT19 := FALSE;
   STATUS[337].EXT.BIT20 := FALSE;
   STATUS[337].EXT.AlarmSuppressed := FALSE;
   STATUS[337].EXT.AlarmPresent := FALSE;
   STATUS[337].EXT.AlarmFailUnAck := FALSE;
   STATUS[337].Status := 0;
   STATUS[337].TimeStamp := 16#0000;
   STATUS[338].EXT.AlarmWarnUnAck := FALSE;
   STATUS[338].EXT.AckRequired := FALSE;
   STATUS[338].EXT.Maintanence := FALSE;
   STATUS[338].EXT.Operation := FALSE;
   STATUS[338].EXT.Forced := FALSE;
   STATUS[338].EXT.BIT29 := FALSE;
   STATUS[338].EXT.BIT30 := FALSE;
   STATUS[338].EXT.BIT31 := FALSE;
   STATUS[338].EXT.ModeBit1 := FALSE;
   STATUS[338].EXT.ModeBit2 := FALSE;
   STATUS[338].EXT.ModeBit3 := FALSE;
   STATUS[338].EXT.BIT19 := FALSE;
   STATUS[338].EXT.BIT20 := FALSE;
   STATUS[338].EXT.AlarmSuppressed := FALSE;
   STATUS[338].EXT.AlarmPresent := FALSE;
   STATUS[338].EXT.AlarmFailUnAck := FALSE;
   STATUS[338].Status := 0;
   STATUS[338].TimeStamp := 16#0000;
   STATUS[339].EXT.AlarmWarnUnAck := FALSE;
   STATUS[339].EXT.AckRequired := FALSE;
   STATUS[339].EXT.Maintanence := FALSE;
   STATUS[339].EXT.Operation := FALSE;
   STATUS[339].EXT.Forced := FALSE;
   STATUS[339].EXT.BIT29 := FALSE;
   STATUS[339].EXT.BIT30 := FALSE;
   STATUS[339].EXT.BIT31 := FALSE;
   STATUS[339].EXT.ModeBit1 := FALSE;
   STATUS[339].EXT.ModeBit2 := FALSE;
   STATUS[339].EXT.ModeBit3 := FALSE;
   STATUS[339].EXT.BIT19 := FALSE;
   STATUS[339].EXT.BIT20 := FALSE;
   STATUS[339].EXT.AlarmSuppressed := FALSE;
   STATUS[339].EXT.AlarmPresent := FALSE;
   STATUS[339].EXT.AlarmFailUnAck := FALSE;
   STATUS[339].Status := 0;
   STATUS[339].TimeStamp := 16#0000;
   STATUS[340].EXT.AlarmWarnUnAck := FALSE;
   STATUS[340].EXT.AckRequired := FALSE;
   STATUS[340].EXT.Maintanence := FALSE;
   STATUS[340].EXT.Operation := FALSE;
   STATUS[340].EXT.Forced := FALSE;
   STATUS[340].EXT.BIT29 := FALSE;
   STATUS[340].EXT.BIT30 := FALSE;
   STATUS[340].EXT.BIT31 := FALSE;
   STATUS[340].EXT.ModeBit1 := FALSE;
   STATUS[340].EXT.ModeBit2 := FALSE;
   STATUS[340].EXT.ModeBit3 := FALSE;
   STATUS[340].EXT.BIT19 := FALSE;
   STATUS[340].EXT.BIT20 := FALSE;
   STATUS[340].EXT.AlarmSuppressed := FALSE;
   STATUS[340].EXT.AlarmPresent := FALSE;
   STATUS[340].EXT.AlarmFailUnAck := FALSE;
   STATUS[340].Status := 0;
   STATUS[340].TimeStamp := 16#0000;
   STATUS[341].EXT.AlarmWarnUnAck := FALSE;
   STATUS[341].EXT.AckRequired := FALSE;
   STATUS[341].EXT.Maintanence := FALSE;
   STATUS[341].EXT.Operation := FALSE;
   STATUS[341].EXT.Forced := FALSE;
   STATUS[341].EXT.BIT29 := FALSE;
   STATUS[341].EXT.BIT30 := FALSE;
   STATUS[341].EXT.BIT31 := FALSE;
   STATUS[341].EXT.ModeBit1 := FALSE;
   STATUS[341].EXT.ModeBit2 := FALSE;
   STATUS[341].EXT.ModeBit3 := FALSE;
   STATUS[341].EXT.BIT19 := FALSE;
   STATUS[341].EXT.BIT20 := FALSE;
   STATUS[341].EXT.AlarmSuppressed := FALSE;
   STATUS[341].EXT.AlarmPresent := FALSE;
   STATUS[341].EXT.AlarmFailUnAck := FALSE;
   STATUS[341].Status := 0;
   STATUS[341].TimeStamp := 16#0000;
   STATUS[342].EXT.AlarmWarnUnAck := FALSE;
   STATUS[342].EXT.AckRequired := FALSE;
   STATUS[342].EXT.Maintanence := FALSE;
   STATUS[342].EXT.Operation := FALSE;
   STATUS[342].EXT.Forced := FALSE;
   STATUS[342].EXT.BIT29 := FALSE;
   STATUS[342].EXT.BIT30 := FALSE;
   STATUS[342].EXT.BIT31 := FALSE;
   STATUS[342].EXT.ModeBit1 := FALSE;
   STATUS[342].EXT.ModeBit2 := FALSE;
   STATUS[342].EXT.ModeBit3 := FALSE;
   STATUS[342].EXT.BIT19 := FALSE;
   STATUS[342].EXT.BIT20 := FALSE;
   STATUS[342].EXT.AlarmSuppressed := FALSE;
   STATUS[342].EXT.AlarmPresent := FALSE;
   STATUS[342].EXT.AlarmFailUnAck := FALSE;
   STATUS[342].Status := 0;
   STATUS[342].TimeStamp := 16#0000;
   STATUS[343].EXT.AlarmWarnUnAck := FALSE;
   STATUS[343].EXT.AckRequired := FALSE;
   STATUS[343].EXT.Maintanence := FALSE;
   STATUS[343].EXT.Operation := FALSE;
   STATUS[343].EXT.Forced := FALSE;
   STATUS[343].EXT.BIT29 := FALSE;
   STATUS[343].EXT.BIT30 := FALSE;
   STATUS[343].EXT.BIT31 := FALSE;
   STATUS[343].EXT.ModeBit1 := FALSE;
   STATUS[343].EXT.ModeBit2 := FALSE;
   STATUS[343].EXT.ModeBit3 := FALSE;
   STATUS[343].EXT.BIT19 := FALSE;
   STATUS[343].EXT.BIT20 := FALSE;
   STATUS[343].EXT.AlarmSuppressed := FALSE;
   STATUS[343].EXT.AlarmPresent := FALSE;
   STATUS[343].EXT.AlarmFailUnAck := FALSE;
   STATUS[343].Status := 0;
   STATUS[343].TimeStamp := 16#0000;
   STATUS[344].EXT.AlarmWarnUnAck := FALSE;
   STATUS[344].EXT.AckRequired := FALSE;
   STATUS[344].EXT.Maintanence := FALSE;
   STATUS[344].EXT.Operation := FALSE;
   STATUS[344].EXT.Forced := FALSE;
   STATUS[344].EXT.BIT29 := FALSE;
   STATUS[344].EXT.BIT30 := FALSE;
   STATUS[344].EXT.BIT31 := FALSE;
   STATUS[344].EXT.ModeBit1 := FALSE;
   STATUS[344].EXT.ModeBit2 := FALSE;
   STATUS[344].EXT.ModeBit3 := FALSE;
   STATUS[344].EXT.BIT19 := FALSE;
   STATUS[344].EXT.BIT20 := FALSE;
   STATUS[344].EXT.AlarmSuppressed := FALSE;
   STATUS[344].EXT.AlarmPresent := FALSE;
   STATUS[344].EXT.AlarmFailUnAck := FALSE;
   STATUS[344].Status := 0;
   STATUS[344].TimeStamp := 16#0000;
   STATUS[345].EXT.AlarmWarnUnAck := FALSE;
   STATUS[345].EXT.AckRequired := FALSE;
   STATUS[345].EXT.Maintanence := FALSE;
   STATUS[345].EXT.Operation := FALSE;
   STATUS[345].EXT.Forced := FALSE;
   STATUS[345].EXT.BIT29 := FALSE;
   STATUS[345].EXT.BIT30 := FALSE;
   STATUS[345].EXT.BIT31 := FALSE;
   STATUS[345].EXT.ModeBit1 := FALSE;
   STATUS[345].EXT.ModeBit2 := FALSE;
   STATUS[345].EXT.ModeBit3 := FALSE;
   STATUS[345].EXT.BIT19 := FALSE;
   STATUS[345].EXT.BIT20 := FALSE;
   STATUS[345].EXT.AlarmSuppressed := FALSE;
   STATUS[345].EXT.AlarmPresent := FALSE;
   STATUS[345].EXT.AlarmFailUnAck := FALSE;
   STATUS[345].Status := 0;
   STATUS[345].TimeStamp := 16#0000;
   STATUS[346].EXT.AlarmWarnUnAck := FALSE;
   STATUS[346].EXT.AckRequired := FALSE;
   STATUS[346].EXT.Maintanence := FALSE;
   STATUS[346].EXT.Operation := FALSE;
   STATUS[346].EXT.Forced := FALSE;
   STATUS[346].EXT.BIT29 := FALSE;
   STATUS[346].EXT.BIT30 := FALSE;
   STATUS[346].EXT.BIT31 := FALSE;
   STATUS[346].EXT.ModeBit1 := FALSE;
   STATUS[346].EXT.ModeBit2 := FALSE;
   STATUS[346].EXT.ModeBit3 := FALSE;
   STATUS[346].EXT.BIT19 := FALSE;
   STATUS[346].EXT.BIT20 := FALSE;
   STATUS[346].EXT.AlarmSuppressed := FALSE;
   STATUS[346].EXT.AlarmPresent := FALSE;
   STATUS[346].EXT.AlarmFailUnAck := FALSE;
   STATUS[346].Status := 0;
   STATUS[346].TimeStamp := 16#0000;
   STATUS[347].EXT.AlarmWarnUnAck := FALSE;
   STATUS[347].EXT.AckRequired := FALSE;
   STATUS[347].EXT.Maintanence := FALSE;
   STATUS[347].EXT.Operation := FALSE;
   STATUS[347].EXT.Forced := FALSE;
   STATUS[347].EXT.BIT29 := FALSE;
   STATUS[347].EXT.BIT30 := FALSE;
   STATUS[347].EXT.BIT31 := FALSE;
   STATUS[347].EXT.ModeBit1 := FALSE;
   STATUS[347].EXT.ModeBit2 := FALSE;
   STATUS[347].EXT.ModeBit3 := FALSE;
   STATUS[347].EXT.BIT19 := FALSE;
   STATUS[347].EXT.BIT20 := FALSE;
   STATUS[347].EXT.AlarmSuppressed := FALSE;
   STATUS[347].EXT.AlarmPresent := FALSE;
   STATUS[347].EXT.AlarmFailUnAck := FALSE;
   STATUS[347].Status := 0;
   STATUS[347].TimeStamp := 16#0000;
   STATUS[348].EXT.AlarmWarnUnAck := FALSE;
   STATUS[348].EXT.AckRequired := FALSE;
   STATUS[348].EXT.Maintanence := FALSE;
   STATUS[348].EXT.Operation := FALSE;
   STATUS[348].EXT.Forced := FALSE;
   STATUS[348].EXT.BIT29 := FALSE;
   STATUS[348].EXT.BIT30 := FALSE;
   STATUS[348].EXT.BIT31 := FALSE;
   STATUS[348].EXT.ModeBit1 := FALSE;
   STATUS[348].EXT.ModeBit2 := FALSE;
   STATUS[348].EXT.ModeBit3 := FALSE;
   STATUS[348].EXT.BIT19 := FALSE;
   STATUS[348].EXT.BIT20 := FALSE;
   STATUS[348].EXT.AlarmSuppressed := FALSE;
   STATUS[348].EXT.AlarmPresent := FALSE;
   STATUS[348].EXT.AlarmFailUnAck := FALSE;
   STATUS[348].Status := 0;
   STATUS[348].TimeStamp := 16#0000;
   STATUS[349].EXT.AlarmWarnUnAck := FALSE;
   STATUS[349].EXT.AckRequired := FALSE;
   STATUS[349].EXT.Maintanence := FALSE;
   STATUS[349].EXT.Operation := FALSE;
   STATUS[349].EXT.Forced := FALSE;
   STATUS[349].EXT.BIT29 := FALSE;
   STATUS[349].EXT.BIT30 := FALSE;
   STATUS[349].EXT.BIT31 := FALSE;
   STATUS[349].EXT.ModeBit1 := FALSE;
   STATUS[349].EXT.ModeBit2 := FALSE;
   STATUS[349].EXT.ModeBit3 := FALSE;
   STATUS[349].EXT.BIT19 := FALSE;
   STATUS[349].EXT.BIT20 := FALSE;
   STATUS[349].EXT.AlarmSuppressed := FALSE;
   STATUS[349].EXT.AlarmPresent := FALSE;
   STATUS[349].EXT.AlarmFailUnAck := FALSE;
   STATUS[349].Status := 0;
   STATUS[349].TimeStamp := 16#0000;
   STATUS[350].EXT.AlarmWarnUnAck := FALSE;
   STATUS[350].EXT.AckRequired := FALSE;
   STATUS[350].EXT.Maintanence := FALSE;
   STATUS[350].EXT.Operation := FALSE;
   STATUS[350].EXT.Forced := FALSE;
   STATUS[350].EXT.BIT29 := FALSE;
   STATUS[350].EXT.BIT30 := FALSE;
   STATUS[350].EXT.BIT31 := FALSE;
   STATUS[350].EXT.ModeBit1 := FALSE;
   STATUS[350].EXT.ModeBit2 := FALSE;
   STATUS[350].EXT.ModeBit3 := FALSE;
   STATUS[350].EXT.BIT19 := FALSE;
   STATUS[350].EXT.BIT20 := FALSE;
   STATUS[350].EXT.AlarmSuppressed := FALSE;
   STATUS[350].EXT.AlarmPresent := FALSE;
   STATUS[350].EXT.AlarmFailUnAck := FALSE;
   STATUS[350].Status := 0;
   STATUS[350].TimeStamp := 16#0000;
   STATUS[351].EXT.AlarmWarnUnAck := FALSE;
   STATUS[351].EXT.AckRequired := FALSE;
   STATUS[351].EXT.Maintanence := FALSE;
   STATUS[351].EXT.Operation := FALSE;
   STATUS[351].EXT.Forced := FALSE;
   STATUS[351].EXT.BIT29 := FALSE;
   STATUS[351].EXT.BIT30 := FALSE;
   STATUS[351].EXT.BIT31 := FALSE;
   STATUS[351].EXT.ModeBit1 := FALSE;
   STATUS[351].EXT.ModeBit2 := FALSE;
   STATUS[351].EXT.ModeBit3 := FALSE;
   STATUS[351].EXT.BIT19 := FALSE;
   STATUS[351].EXT.BIT20 := FALSE;
   STATUS[351].EXT.AlarmSuppressed := FALSE;
   STATUS[351].EXT.AlarmPresent := FALSE;
   STATUS[351].EXT.AlarmFailUnAck := FALSE;
   STATUS[351].Status := 0;
   STATUS[351].TimeStamp := 16#0000;
   STATUS[352].EXT.AlarmWarnUnAck := FALSE;
   STATUS[352].EXT.AckRequired := FALSE;
   STATUS[352].EXT.Maintanence := FALSE;
   STATUS[352].EXT.Operation := FALSE;
   STATUS[352].EXT.Forced := FALSE;
   STATUS[352].EXT.BIT29 := FALSE;
   STATUS[352].EXT.BIT30 := FALSE;
   STATUS[352].EXT.BIT31 := FALSE;
   STATUS[352].EXT.ModeBit1 := FALSE;
   STATUS[352].EXT.ModeBit2 := FALSE;
   STATUS[352].EXT.ModeBit3 := FALSE;
   STATUS[352].EXT.BIT19 := FALSE;
   STATUS[352].EXT.BIT20 := FALSE;
   STATUS[352].EXT.AlarmSuppressed := FALSE;
   STATUS[352].EXT.AlarmPresent := FALSE;
   STATUS[352].EXT.AlarmFailUnAck := FALSE;
   STATUS[352].Status := 0;
   STATUS[352].TimeStamp := 16#0000;
   STATUS[353].EXT.AlarmWarnUnAck := FALSE;
   STATUS[353].EXT.AckRequired := FALSE;
   STATUS[353].EXT.Maintanence := FALSE;
   STATUS[353].EXT.Operation := FALSE;
   STATUS[353].EXT.Forced := FALSE;
   STATUS[353].EXT.BIT29 := FALSE;
   STATUS[353].EXT.BIT30 := FALSE;
   STATUS[353].EXT.BIT31 := FALSE;
   STATUS[353].EXT.ModeBit1 := FALSE;
   STATUS[353].EXT.ModeBit2 := FALSE;
   STATUS[353].EXT.ModeBit3 := FALSE;
   STATUS[353].EXT.BIT19 := FALSE;
   STATUS[353].EXT.BIT20 := FALSE;
   STATUS[353].EXT.AlarmSuppressed := FALSE;
   STATUS[353].EXT.AlarmPresent := FALSE;
   STATUS[353].EXT.AlarmFailUnAck := FALSE;
   STATUS[353].Status := 0;
   STATUS[353].TimeStamp := 16#0000;
   STATUS[354].EXT.AlarmWarnUnAck := FALSE;
   STATUS[354].EXT.AckRequired := FALSE;
   STATUS[354].EXT.Maintanence := FALSE;
   STATUS[354].EXT.Operation := FALSE;
   STATUS[354].EXT.Forced := FALSE;
   STATUS[354].EXT.BIT29 := FALSE;
   STATUS[354].EXT.BIT30 := FALSE;
   STATUS[354].EXT.BIT31 := FALSE;
   STATUS[354].EXT.ModeBit1 := FALSE;
   STATUS[354].EXT.ModeBit2 := FALSE;
   STATUS[354].EXT.ModeBit3 := FALSE;
   STATUS[354].EXT.BIT19 := FALSE;
   STATUS[354].EXT.BIT20 := FALSE;
   STATUS[354].EXT.AlarmSuppressed := FALSE;
   STATUS[354].EXT.AlarmPresent := FALSE;
   STATUS[354].EXT.AlarmFailUnAck := FALSE;
   STATUS[354].Status := 0;
   STATUS[354].TimeStamp := 16#0000;
   STATUS[355].EXT.AlarmWarnUnAck := FALSE;
   STATUS[355].EXT.AckRequired := FALSE;
   STATUS[355].EXT.Maintanence := FALSE;
   STATUS[355].EXT.Operation := FALSE;
   STATUS[355].EXT.Forced := FALSE;
   STATUS[355].EXT.BIT29 := FALSE;
   STATUS[355].EXT.BIT30 := FALSE;
   STATUS[355].EXT.BIT31 := FALSE;
   STATUS[355].EXT.ModeBit1 := FALSE;
   STATUS[355].EXT.ModeBit2 := FALSE;
   STATUS[355].EXT.ModeBit3 := FALSE;
   STATUS[355].EXT.BIT19 := FALSE;
   STATUS[355].EXT.BIT20 := FALSE;
   STATUS[355].EXT.AlarmSuppressed := FALSE;
   STATUS[355].EXT.AlarmPresent := FALSE;
   STATUS[355].EXT.AlarmFailUnAck := FALSE;
   STATUS[355].Status := 0;
   STATUS[355].TimeStamp := 16#0000;
   STATUS[356].EXT.AlarmWarnUnAck := FALSE;
   STATUS[356].EXT.AckRequired := FALSE;
   STATUS[356].EXT.Maintanence := FALSE;
   STATUS[356].EXT.Operation := FALSE;
   STATUS[356].EXT.Forced := FALSE;
   STATUS[356].EXT.BIT29 := FALSE;
   STATUS[356].EXT.BIT30 := FALSE;
   STATUS[356].EXT.BIT31 := FALSE;
   STATUS[356].EXT.ModeBit1 := FALSE;
   STATUS[356].EXT.ModeBit2 := FALSE;
   STATUS[356].EXT.ModeBit3 := FALSE;
   STATUS[356].EXT.BIT19 := FALSE;
   STATUS[356].EXT.BIT20 := FALSE;
   STATUS[356].EXT.AlarmSuppressed := FALSE;
   STATUS[356].EXT.AlarmPresent := FALSE;
   STATUS[356].EXT.AlarmFailUnAck := FALSE;
   STATUS[356].Status := 0;
   STATUS[356].TimeStamp := 16#0000;
   STATUS[357].EXT.AlarmWarnUnAck := FALSE;
   STATUS[357].EXT.AckRequired := FALSE;
   STATUS[357].EXT.Maintanence := FALSE;
   STATUS[357].EXT.Operation := FALSE;
   STATUS[357].EXT.Forced := FALSE;
   STATUS[357].EXT.BIT29 := FALSE;
   STATUS[357].EXT.BIT30 := FALSE;
   STATUS[357].EXT.BIT31 := FALSE;
   STATUS[357].EXT.ModeBit1 := FALSE;
   STATUS[357].EXT.ModeBit2 := FALSE;
   STATUS[357].EXT.ModeBit3 := FALSE;
   STATUS[357].EXT.BIT19 := FALSE;
   STATUS[357].EXT.BIT20 := FALSE;
   STATUS[357].EXT.AlarmSuppressed := FALSE;
   STATUS[357].EXT.AlarmPresent := FALSE;
   STATUS[357].EXT.AlarmFailUnAck := FALSE;
   STATUS[357].Status := 0;
   STATUS[357].TimeStamp := 16#0000;
   STATUS[358].EXT.AlarmWarnUnAck := FALSE;
   STATUS[358].EXT.AckRequired := FALSE;
   STATUS[358].EXT.Maintanence := FALSE;
   STATUS[358].EXT.Operation := FALSE;
   STATUS[358].EXT.Forced := FALSE;
   STATUS[358].EXT.BIT29 := FALSE;
   STATUS[358].EXT.BIT30 := FALSE;
   STATUS[358].EXT.BIT31 := FALSE;
   STATUS[358].EXT.ModeBit1 := FALSE;
   STATUS[358].EXT.ModeBit2 := FALSE;
   STATUS[358].EXT.ModeBit3 := FALSE;
   STATUS[358].EXT.BIT19 := FALSE;
   STATUS[358].EXT.BIT20 := FALSE;
   STATUS[358].EXT.AlarmSuppressed := FALSE;
   STATUS[358].EXT.AlarmPresent := FALSE;
   STATUS[358].EXT.AlarmFailUnAck := FALSE;
   STATUS[358].Status := 0;
   STATUS[358].TimeStamp := 16#0000;
   STATUS[359].EXT.AlarmWarnUnAck := FALSE;
   STATUS[359].EXT.AckRequired := FALSE;
   STATUS[359].EXT.Maintanence := FALSE;
   STATUS[359].EXT.Operation := FALSE;
   STATUS[359].EXT.Forced := FALSE;
   STATUS[359].EXT.BIT29 := FALSE;
   STATUS[359].EXT.BIT30 := FALSE;
   STATUS[359].EXT.BIT31 := FALSE;
   STATUS[359].EXT.ModeBit1 := FALSE;
   STATUS[359].EXT.ModeBit2 := FALSE;
   STATUS[359].EXT.ModeBit3 := FALSE;
   STATUS[359].EXT.BIT19 := FALSE;
   STATUS[359].EXT.BIT20 := FALSE;
   STATUS[359].EXT.AlarmSuppressed := FALSE;
   STATUS[359].EXT.AlarmPresent := FALSE;
   STATUS[359].EXT.AlarmFailUnAck := FALSE;
   STATUS[359].Status := 0;
   STATUS[359].TimeStamp := 16#0000;
   STATUS[360].EXT.AlarmWarnUnAck := FALSE;
   STATUS[360].EXT.AckRequired := FALSE;
   STATUS[360].EXT.Maintanence := FALSE;
   STATUS[360].EXT.Operation := FALSE;
   STATUS[360].EXT.Forced := FALSE;
   STATUS[360].EXT.BIT29 := FALSE;
   STATUS[360].EXT.BIT30 := FALSE;
   STATUS[360].EXT.BIT31 := FALSE;
   STATUS[360].EXT.ModeBit1 := FALSE;
   STATUS[360].EXT.ModeBit2 := FALSE;
   STATUS[360].EXT.ModeBit3 := FALSE;
   STATUS[360].EXT.BIT19 := FALSE;
   STATUS[360].EXT.BIT20 := FALSE;
   STATUS[360].EXT.AlarmSuppressed := FALSE;
   STATUS[360].EXT.AlarmPresent := FALSE;
   STATUS[360].EXT.AlarmFailUnAck := FALSE;
   STATUS[360].Status := 0;
   STATUS[360].TimeStamp := 16#0000;
   STATUS[361].EXT.AlarmWarnUnAck := FALSE;
   STATUS[361].EXT.AckRequired := FALSE;
   STATUS[361].EXT.Maintanence := FALSE;
   STATUS[361].EXT.Operation := FALSE;
   STATUS[361].EXT.Forced := FALSE;
   STATUS[361].EXT.BIT29 := FALSE;
   STATUS[361].EXT.BIT30 := FALSE;
   STATUS[361].EXT.BIT31 := FALSE;
   STATUS[361].EXT.ModeBit1 := FALSE;
   STATUS[361].EXT.ModeBit2 := FALSE;
   STATUS[361].EXT.ModeBit3 := FALSE;
   STATUS[361].EXT.BIT19 := FALSE;
   STATUS[361].EXT.BIT20 := FALSE;
   STATUS[361].EXT.AlarmSuppressed := FALSE;
   STATUS[361].EXT.AlarmPresent := FALSE;
   STATUS[361].EXT.AlarmFailUnAck := FALSE;
   STATUS[361].Status := 0;
   STATUS[361].TimeStamp := 16#0000;
   STATUS[362].EXT.AlarmWarnUnAck := FALSE;
   STATUS[362].EXT.AckRequired := FALSE;
   STATUS[362].EXT.Maintanence := FALSE;
   STATUS[362].EXT.Operation := FALSE;
   STATUS[362].EXT.Forced := FALSE;
   STATUS[362].EXT.BIT29 := FALSE;
   STATUS[362].EXT.BIT30 := FALSE;
   STATUS[362].EXT.BIT31 := FALSE;
   STATUS[362].EXT.ModeBit1 := FALSE;
   STATUS[362].EXT.ModeBit2 := FALSE;
   STATUS[362].EXT.ModeBit3 := FALSE;
   STATUS[362].EXT.BIT19 := FALSE;
   STATUS[362].EXT.BIT20 := FALSE;
   STATUS[362].EXT.AlarmSuppressed := FALSE;
   STATUS[362].EXT.AlarmPresent := FALSE;
   STATUS[362].EXT.AlarmFailUnAck := FALSE;
   STATUS[362].Status := 0;
   STATUS[362].TimeStamp := 16#0000;
   STATUS[363].EXT.AlarmWarnUnAck := FALSE;
   STATUS[363].EXT.AckRequired := FALSE;
   STATUS[363].EXT.Maintanence := FALSE;
   STATUS[363].EXT.Operation := FALSE;
   STATUS[363].EXT.Forced := FALSE;
   STATUS[363].EXT.BIT29 := FALSE;
   STATUS[363].EXT.BIT30 := FALSE;
   STATUS[363].EXT.BIT31 := FALSE;
   STATUS[363].EXT.ModeBit1 := FALSE;
   STATUS[363].EXT.ModeBit2 := FALSE;
   STATUS[363].EXT.ModeBit3 := FALSE;
   STATUS[363].EXT.BIT19 := FALSE;
   STATUS[363].EXT.BIT20 := FALSE;
   STATUS[363].EXT.AlarmSuppressed := FALSE;
   STATUS[363].EXT.AlarmPresent := FALSE;
   STATUS[363].EXT.AlarmFailUnAck := FALSE;
   STATUS[363].Status := 0;
   STATUS[363].TimeStamp := 16#0000;
   STATUS[364].EXT.AlarmWarnUnAck := FALSE;
   STATUS[364].EXT.AckRequired := FALSE;
   STATUS[364].EXT.Maintanence := FALSE;
   STATUS[364].EXT.Operation := FALSE;
   STATUS[364].EXT.Forced := FALSE;
   STATUS[364].EXT.BIT29 := FALSE;
   STATUS[364].EXT.BIT30 := FALSE;
   STATUS[364].EXT.BIT31 := FALSE;
   STATUS[364].EXT.ModeBit1 := FALSE;
   STATUS[364].EXT.ModeBit2 := FALSE;
   STATUS[364].EXT.ModeBit3 := FALSE;
   STATUS[364].EXT.BIT19 := FALSE;
   STATUS[364].EXT.BIT20 := FALSE;
   STATUS[364].EXT.AlarmSuppressed := FALSE;
   STATUS[364].EXT.AlarmPresent := FALSE;
   STATUS[364].EXT.AlarmFailUnAck := FALSE;
   STATUS[364].Status := 0;
   STATUS[364].TimeStamp := 16#0000;
   STATUS[365].EXT.AlarmWarnUnAck := FALSE;
   STATUS[365].EXT.AckRequired := FALSE;
   STATUS[365].EXT.Maintanence := FALSE;
   STATUS[365].EXT.Operation := FALSE;
   STATUS[365].EXT.Forced := FALSE;
   STATUS[365].EXT.BIT29 := FALSE;
   STATUS[365].EXT.BIT30 := FALSE;
   STATUS[365].EXT.BIT31 := FALSE;
   STATUS[365].EXT.ModeBit1 := FALSE;
   STATUS[365].EXT.ModeBit2 := FALSE;
   STATUS[365].EXT.ModeBit3 := FALSE;
   STATUS[365].EXT.BIT19 := FALSE;
   STATUS[365].EXT.BIT20 := FALSE;
   STATUS[365].EXT.AlarmSuppressed := FALSE;
   STATUS[365].EXT.AlarmPresent := FALSE;
   STATUS[365].EXT.AlarmFailUnAck := FALSE;
   STATUS[365].Status := 0;
   STATUS[365].TimeStamp := 16#0000;
   STATUS[366].EXT.AlarmWarnUnAck := FALSE;
   STATUS[366].EXT.AckRequired := FALSE;
   STATUS[366].EXT.Maintanence := FALSE;
   STATUS[366].EXT.Operation := FALSE;
   STATUS[366].EXT.Forced := FALSE;
   STATUS[366].EXT.BIT29 := FALSE;
   STATUS[366].EXT.BIT30 := FALSE;
   STATUS[366].EXT.BIT31 := FALSE;
   STATUS[366].EXT.ModeBit1 := FALSE;
   STATUS[366].EXT.ModeBit2 := FALSE;
   STATUS[366].EXT.ModeBit3 := FALSE;
   STATUS[366].EXT.BIT19 := FALSE;
   STATUS[366].EXT.BIT20 := FALSE;
   STATUS[366].EXT.AlarmSuppressed := FALSE;
   STATUS[366].EXT.AlarmPresent := FALSE;
   STATUS[366].EXT.AlarmFailUnAck := FALSE;
   STATUS[366].Status := 0;
   STATUS[366].TimeStamp := 16#0000;
   STATUS[367].EXT.AlarmWarnUnAck := FALSE;
   STATUS[367].EXT.AckRequired := FALSE;
   STATUS[367].EXT.Maintanence := FALSE;
   STATUS[367].EXT.Operation := FALSE;
   STATUS[367].EXT.Forced := FALSE;
   STATUS[367].EXT.BIT29 := FALSE;
   STATUS[367].EXT.BIT30 := FALSE;
   STATUS[367].EXT.BIT31 := FALSE;
   STATUS[367].EXT.ModeBit1 := FALSE;
   STATUS[367].EXT.ModeBit2 := FALSE;
   STATUS[367].EXT.ModeBit3 := FALSE;
   STATUS[367].EXT.BIT19 := FALSE;
   STATUS[367].EXT.BIT20 := FALSE;
   STATUS[367].EXT.AlarmSuppressed := FALSE;
   STATUS[367].EXT.AlarmPresent := FALSE;
   STATUS[367].EXT.AlarmFailUnAck := FALSE;
   STATUS[367].Status := 0;
   STATUS[367].TimeStamp := 16#0000;
   STATUS[368].EXT.AlarmWarnUnAck := FALSE;
   STATUS[368].EXT.AckRequired := FALSE;
   STATUS[368].EXT.Maintanence := FALSE;
   STATUS[368].EXT.Operation := FALSE;
   STATUS[368].EXT.Forced := FALSE;
   STATUS[368].EXT.BIT29 := FALSE;
   STATUS[368].EXT.BIT30 := FALSE;
   STATUS[368].EXT.BIT31 := FALSE;
   STATUS[368].EXT.ModeBit1 := FALSE;
   STATUS[368].EXT.ModeBit2 := FALSE;
   STATUS[368].EXT.ModeBit3 := FALSE;
   STATUS[368].EXT.BIT19 := FALSE;
   STATUS[368].EXT.BIT20 := FALSE;
   STATUS[368].EXT.AlarmSuppressed := FALSE;
   STATUS[368].EXT.AlarmPresent := FALSE;
   STATUS[368].EXT.AlarmFailUnAck := FALSE;
   STATUS[368].Status := 0;
   STATUS[368].TimeStamp := 16#0000;
   STATUS[369].EXT.AlarmWarnUnAck := FALSE;
   STATUS[369].EXT.AckRequired := FALSE;
   STATUS[369].EXT.Maintanence := FALSE;
   STATUS[369].EXT.Operation := FALSE;
   STATUS[369].EXT.Forced := FALSE;
   STATUS[369].EXT.BIT29 := FALSE;
   STATUS[369].EXT.BIT30 := FALSE;
   STATUS[369].EXT.BIT31 := FALSE;
   STATUS[369].EXT.ModeBit1 := FALSE;
   STATUS[369].EXT.ModeBit2 := FALSE;
   STATUS[369].EXT.ModeBit3 := FALSE;
   STATUS[369].EXT.BIT19 := FALSE;
   STATUS[369].EXT.BIT20 := FALSE;
   STATUS[369].EXT.AlarmSuppressed := FALSE;
   STATUS[369].EXT.AlarmPresent := FALSE;
   STATUS[369].EXT.AlarmFailUnAck := FALSE;
   STATUS[369].Status := 0;
   STATUS[369].TimeStamp := 16#0000;
   STATUS[370].EXT.AlarmWarnUnAck := FALSE;
   STATUS[370].EXT.AckRequired := FALSE;
   STATUS[370].EXT.Maintanence := FALSE;
   STATUS[370].EXT.Operation := FALSE;
   STATUS[370].EXT.Forced := FALSE;
   STATUS[370].EXT.BIT29 := FALSE;
   STATUS[370].EXT.BIT30 := FALSE;
   STATUS[370].EXT.BIT31 := FALSE;
   STATUS[370].EXT.ModeBit1 := FALSE;
   STATUS[370].EXT.ModeBit2 := FALSE;
   STATUS[370].EXT.ModeBit3 := FALSE;
   STATUS[370].EXT.BIT19 := FALSE;
   STATUS[370].EXT.BIT20 := FALSE;
   STATUS[370].EXT.AlarmSuppressed := FALSE;
   STATUS[370].EXT.AlarmPresent := FALSE;
   STATUS[370].EXT.AlarmFailUnAck := FALSE;
   STATUS[370].Status := 0;
   STATUS[370].TimeStamp := 16#0000;
   STATUS[371].EXT.AlarmWarnUnAck := FALSE;
   STATUS[371].EXT.AckRequired := FALSE;
   STATUS[371].EXT.Maintanence := FALSE;
   STATUS[371].EXT.Operation := FALSE;
   STATUS[371].EXT.Forced := FALSE;
   STATUS[371].EXT.BIT29 := FALSE;
   STATUS[371].EXT.BIT30 := FALSE;
   STATUS[371].EXT.BIT31 := FALSE;
   STATUS[371].EXT.ModeBit1 := FALSE;
   STATUS[371].EXT.ModeBit2 := FALSE;
   STATUS[371].EXT.ModeBit3 := FALSE;
   STATUS[371].EXT.BIT19 := FALSE;
   STATUS[371].EXT.BIT20 := FALSE;
   STATUS[371].EXT.AlarmSuppressed := FALSE;
   STATUS[371].EXT.AlarmPresent := FALSE;
   STATUS[371].EXT.AlarmFailUnAck := FALSE;
   STATUS[371].Status := 0;
   STATUS[371].TimeStamp := 16#0000;
   STATUS[372].EXT.AlarmWarnUnAck := FALSE;
   STATUS[372].EXT.AckRequired := FALSE;
   STATUS[372].EXT.Maintanence := FALSE;
   STATUS[372].EXT.Operation := FALSE;
   STATUS[372].EXT.Forced := FALSE;
   STATUS[372].EXT.BIT29 := FALSE;
   STATUS[372].EXT.BIT30 := FALSE;
   STATUS[372].EXT.BIT31 := FALSE;
   STATUS[372].EXT.ModeBit1 := FALSE;
   STATUS[372].EXT.ModeBit2 := FALSE;
   STATUS[372].EXT.ModeBit3 := FALSE;
   STATUS[372].EXT.BIT19 := FALSE;
   STATUS[372].EXT.BIT20 := FALSE;
   STATUS[372].EXT.AlarmSuppressed := FALSE;
   STATUS[372].EXT.AlarmPresent := FALSE;
   STATUS[372].EXT.AlarmFailUnAck := FALSE;
   STATUS[372].Status := 0;
   STATUS[372].TimeStamp := 16#0000;
   STATUS[373].EXT.AlarmWarnUnAck := FALSE;
   STATUS[373].EXT.AckRequired := FALSE;
   STATUS[373].EXT.Maintanence := FALSE;
   STATUS[373].EXT.Operation := FALSE;
   STATUS[373].EXT.Forced := FALSE;
   STATUS[373].EXT.BIT29 := FALSE;
   STATUS[373].EXT.BIT30 := FALSE;
   STATUS[373].EXT.BIT31 := FALSE;
   STATUS[373].EXT.ModeBit1 := FALSE;
   STATUS[373].EXT.ModeBit2 := FALSE;
   STATUS[373].EXT.ModeBit3 := FALSE;
   STATUS[373].EXT.BIT19 := FALSE;
   STATUS[373].EXT.BIT20 := FALSE;
   STATUS[373].EXT.AlarmSuppressed := FALSE;
   STATUS[373].EXT.AlarmPresent := FALSE;
   STATUS[373].EXT.AlarmFailUnAck := FALSE;
   STATUS[373].Status := 0;
   STATUS[373].TimeStamp := 16#0000;
   STATUS[374].EXT.AlarmWarnUnAck := FALSE;
   STATUS[374].EXT.AckRequired := FALSE;
   STATUS[374].EXT.Maintanence := FALSE;
   STATUS[374].EXT.Operation := FALSE;
   STATUS[374].EXT.Forced := FALSE;
   STATUS[374].EXT.BIT29 := FALSE;
   STATUS[374].EXT.BIT30 := FALSE;
   STATUS[374].EXT.BIT31 := FALSE;
   STATUS[374].EXT.ModeBit1 := FALSE;
   STATUS[374].EXT.ModeBit2 := FALSE;
   STATUS[374].EXT.ModeBit3 := FALSE;
   STATUS[374].EXT.BIT19 := FALSE;
   STATUS[374].EXT.BIT20 := FALSE;
   STATUS[374].EXT.AlarmSuppressed := FALSE;
   STATUS[374].EXT.AlarmPresent := FALSE;
   STATUS[374].EXT.AlarmFailUnAck := FALSE;
   STATUS[374].Status := 0;
   STATUS[374].TimeStamp := 16#0000;
   STATUS[375].EXT.AlarmWarnUnAck := FALSE;
   STATUS[375].EXT.AckRequired := FALSE;
   STATUS[375].EXT.Maintanence := FALSE;
   STATUS[375].EXT.Operation := FALSE;
   STATUS[375].EXT.Forced := FALSE;
   STATUS[375].EXT.BIT29 := FALSE;
   STATUS[375].EXT.BIT30 := FALSE;
   STATUS[375].EXT.BIT31 := FALSE;
   STATUS[375].EXT.ModeBit1 := FALSE;
   STATUS[375].EXT.ModeBit2 := FALSE;
   STATUS[375].EXT.ModeBit3 := FALSE;
   STATUS[375].EXT.BIT19 := FALSE;
   STATUS[375].EXT.BIT20 := FALSE;
   STATUS[375].EXT.AlarmSuppressed := FALSE;
   STATUS[375].EXT.AlarmPresent := FALSE;
   STATUS[375].EXT.AlarmFailUnAck := FALSE;
   STATUS[375].Status := 0;
   STATUS[375].TimeStamp := 16#0000;
   STATUS[376].EXT.AlarmWarnUnAck := FALSE;
   STATUS[376].EXT.AckRequired := FALSE;
   STATUS[376].EXT.Maintanence := FALSE;
   STATUS[376].EXT.Operation := FALSE;
   STATUS[376].EXT.Forced := FALSE;
   STATUS[376].EXT.BIT29 := FALSE;
   STATUS[376].EXT.BIT30 := FALSE;
   STATUS[376].EXT.BIT31 := FALSE;
   STATUS[376].EXT.ModeBit1 := FALSE;
   STATUS[376].EXT.ModeBit2 := FALSE;
   STATUS[376].EXT.ModeBit3 := FALSE;
   STATUS[376].EXT.BIT19 := FALSE;
   STATUS[376].EXT.BIT20 := FALSE;
   STATUS[376].EXT.AlarmSuppressed := FALSE;
   STATUS[376].EXT.AlarmPresent := FALSE;
   STATUS[376].EXT.AlarmFailUnAck := FALSE;
   STATUS[376].Status := 0;
   STATUS[376].TimeStamp := 16#0000;
   STATUS[377].EXT.AlarmWarnUnAck := FALSE;
   STATUS[377].EXT.AckRequired := FALSE;
   STATUS[377].EXT.Maintanence := FALSE;
   STATUS[377].EXT.Operation := FALSE;
   STATUS[377].EXT.Forced := FALSE;
   STATUS[377].EXT.BIT29 := FALSE;
   STATUS[377].EXT.BIT30 := FALSE;
   STATUS[377].EXT.BIT31 := FALSE;
   STATUS[377].EXT.ModeBit1 := FALSE;
   STATUS[377].EXT.ModeBit2 := FALSE;
   STATUS[377].EXT.ModeBit3 := FALSE;
   STATUS[377].EXT.BIT19 := FALSE;
   STATUS[377].EXT.BIT20 := FALSE;
   STATUS[377].EXT.AlarmSuppressed := FALSE;
   STATUS[377].EXT.AlarmPresent := FALSE;
   STATUS[377].EXT.AlarmFailUnAck := FALSE;
   STATUS[377].Status := 0;
   STATUS[377].TimeStamp := 16#0000;
   STATUS[378].EXT.AlarmWarnUnAck := FALSE;
   STATUS[378].EXT.AckRequired := FALSE;
   STATUS[378].EXT.Maintanence := FALSE;
   STATUS[378].EXT.Operation := FALSE;
   STATUS[378].EXT.Forced := FALSE;
   STATUS[378].EXT.BIT29 := FALSE;
   STATUS[378].EXT.BIT30 := FALSE;
   STATUS[378].EXT.BIT31 := FALSE;
   STATUS[378].EXT.ModeBit1 := FALSE;
   STATUS[378].EXT.ModeBit2 := FALSE;
   STATUS[378].EXT.ModeBit3 := FALSE;
   STATUS[378].EXT.BIT19 := FALSE;
   STATUS[378].EXT.BIT20 := FALSE;
   STATUS[378].EXT.AlarmSuppressed := FALSE;
   STATUS[378].EXT.AlarmPresent := FALSE;
   STATUS[378].EXT.AlarmFailUnAck := FALSE;
   STATUS[378].Status := 0;
   STATUS[378].TimeStamp := 16#0000;
   STATUS[379].EXT.AlarmWarnUnAck := FALSE;
   STATUS[379].EXT.AckRequired := FALSE;
   STATUS[379].EXT.Maintanence := FALSE;
   STATUS[379].EXT.Operation := FALSE;
   STATUS[379].EXT.Forced := FALSE;
   STATUS[379].EXT.BIT29 := FALSE;
   STATUS[379].EXT.BIT30 := FALSE;
   STATUS[379].EXT.BIT31 := FALSE;
   STATUS[379].EXT.ModeBit1 := FALSE;
   STATUS[379].EXT.ModeBit2 := FALSE;
   STATUS[379].EXT.ModeBit3 := FALSE;
   STATUS[379].EXT.BIT19 := FALSE;
   STATUS[379].EXT.BIT20 := FALSE;
   STATUS[379].EXT.AlarmSuppressed := FALSE;
   STATUS[379].EXT.AlarmPresent := FALSE;
   STATUS[379].EXT.AlarmFailUnAck := FALSE;
   STATUS[379].Status := 0;
   STATUS[379].TimeStamp := 16#0000;
   STATUS[380].EXT.AlarmWarnUnAck := FALSE;
   STATUS[380].EXT.AckRequired := FALSE;
   STATUS[380].EXT.Maintanence := FALSE;
   STATUS[380].EXT.Operation := FALSE;
   STATUS[380].EXT.Forced := FALSE;
   STATUS[380].EXT.BIT29 := FALSE;
   STATUS[380].EXT.BIT30 := FALSE;
   STATUS[380].EXT.BIT31 := FALSE;
   STATUS[380].EXT.ModeBit1 := FALSE;
   STATUS[380].EXT.ModeBit2 := FALSE;
   STATUS[380].EXT.ModeBit3 := FALSE;
   STATUS[380].EXT.BIT19 := FALSE;
   STATUS[380].EXT.BIT20 := FALSE;
   STATUS[380].EXT.AlarmSuppressed := FALSE;
   STATUS[380].EXT.AlarmPresent := FALSE;
   STATUS[380].EXT.AlarmFailUnAck := FALSE;
   STATUS[380].Status := 0;
   STATUS[380].TimeStamp := 16#0000;
   STATUS[381].EXT.AlarmWarnUnAck := FALSE;
   STATUS[381].EXT.AckRequired := FALSE;
   STATUS[381].EXT.Maintanence := FALSE;
   STATUS[381].EXT.Operation := FALSE;
   STATUS[381].EXT.Forced := FALSE;
   STATUS[381].EXT.BIT29 := FALSE;
   STATUS[381].EXT.BIT30 := FALSE;
   STATUS[381].EXT.BIT31 := FALSE;
   STATUS[381].EXT.ModeBit1 := FALSE;
   STATUS[381].EXT.ModeBit2 := FALSE;
   STATUS[381].EXT.ModeBit3 := FALSE;
   STATUS[381].EXT.BIT19 := FALSE;
   STATUS[381].EXT.BIT20 := FALSE;
   STATUS[381].EXT.AlarmSuppressed := FALSE;
   STATUS[381].EXT.AlarmPresent := FALSE;
   STATUS[381].EXT.AlarmFailUnAck := FALSE;
   STATUS[381].Status := 0;
   STATUS[381].TimeStamp := 16#0000;
   STATUS[382].EXT.AlarmWarnUnAck := FALSE;
   STATUS[382].EXT.AckRequired := FALSE;
   STATUS[382].EXT.Maintanence := FALSE;
   STATUS[382].EXT.Operation := FALSE;
   STATUS[382].EXT.Forced := FALSE;
   STATUS[382].EXT.BIT29 := FALSE;
   STATUS[382].EXT.BIT30 := FALSE;
   STATUS[382].EXT.BIT31 := FALSE;
   STATUS[382].EXT.ModeBit1 := FALSE;
   STATUS[382].EXT.ModeBit2 := FALSE;
   STATUS[382].EXT.ModeBit3 := FALSE;
   STATUS[382].EXT.BIT19 := FALSE;
   STATUS[382].EXT.BIT20 := FALSE;
   STATUS[382].EXT.AlarmSuppressed := FALSE;
   STATUS[382].EXT.AlarmPresent := FALSE;
   STATUS[382].EXT.AlarmFailUnAck := FALSE;
   STATUS[382].Status := 0;
   STATUS[382].TimeStamp := 16#0000;
   STATUS[383].EXT.AlarmWarnUnAck := FALSE;
   STATUS[383].EXT.AckRequired := FALSE;
   STATUS[383].EXT.Maintanence := FALSE;
   STATUS[383].EXT.Operation := FALSE;
   STATUS[383].EXT.Forced := FALSE;
   STATUS[383].EXT.BIT29 := FALSE;
   STATUS[383].EXT.BIT30 := FALSE;
   STATUS[383].EXT.BIT31 := FALSE;
   STATUS[383].EXT.ModeBit1 := FALSE;
   STATUS[383].EXT.ModeBit2 := FALSE;
   STATUS[383].EXT.ModeBit3 := FALSE;
   STATUS[383].EXT.BIT19 := FALSE;
   STATUS[383].EXT.BIT20 := FALSE;
   STATUS[383].EXT.AlarmSuppressed := FALSE;
   STATUS[383].EXT.AlarmPresent := FALSE;
   STATUS[383].EXT.AlarmFailUnAck := FALSE;
   STATUS[383].Status := 0;
   STATUS[383].TimeStamp := 16#0000;
   STATUS[384].EXT.AlarmWarnUnAck := FALSE;
   STATUS[384].EXT.AckRequired := FALSE;
   STATUS[384].EXT.Maintanence := FALSE;
   STATUS[384].EXT.Operation := FALSE;
   STATUS[384].EXT.Forced := FALSE;
   STATUS[384].EXT.BIT29 := FALSE;
   STATUS[384].EXT.BIT30 := FALSE;
   STATUS[384].EXT.BIT31 := FALSE;
   STATUS[384].EXT.ModeBit1 := FALSE;
   STATUS[384].EXT.ModeBit2 := FALSE;
   STATUS[384].EXT.ModeBit3 := FALSE;
   STATUS[384].EXT.BIT19 := FALSE;
   STATUS[384].EXT.BIT20 := FALSE;
   STATUS[384].EXT.AlarmSuppressed := FALSE;
   STATUS[384].EXT.AlarmPresent := FALSE;
   STATUS[384].EXT.AlarmFailUnAck := FALSE;
   STATUS[384].Status := 0;
   STATUS[384].TimeStamp := 16#0000;
   STATUS[385].EXT.AlarmWarnUnAck := FALSE;
   STATUS[385].EXT.AckRequired := FALSE;
   STATUS[385].EXT.Maintanence := FALSE;
   STATUS[385].EXT.Operation := FALSE;
   STATUS[385].EXT.Forced := FALSE;
   STATUS[385].EXT.BIT29 := FALSE;
   STATUS[385].EXT.BIT30 := FALSE;
   STATUS[385].EXT.BIT31 := FALSE;
   STATUS[385].EXT.ModeBit1 := FALSE;
   STATUS[385].EXT.ModeBit2 := FALSE;
   STATUS[385].EXT.ModeBit3 := FALSE;
   STATUS[385].EXT.BIT19 := FALSE;
   STATUS[385].EXT.BIT20 := FALSE;
   STATUS[385].EXT.AlarmSuppressed := FALSE;
   STATUS[385].EXT.AlarmPresent := FALSE;
   STATUS[385].EXT.AlarmFailUnAck := FALSE;
   STATUS[385].Status := 0;
   STATUS[385].TimeStamp := 16#0000;
   STATUS[386].EXT.AlarmWarnUnAck := FALSE;
   STATUS[386].EXT.AckRequired := FALSE;
   STATUS[386].EXT.Maintanence := FALSE;
   STATUS[386].EXT.Operation := FALSE;
   STATUS[386].EXT.Forced := FALSE;
   STATUS[386].EXT.BIT29 := FALSE;
   STATUS[386].EXT.BIT30 := FALSE;
   STATUS[386].EXT.BIT31 := FALSE;
   STATUS[386].EXT.ModeBit1 := FALSE;
   STATUS[386].EXT.ModeBit2 := FALSE;
   STATUS[386].EXT.ModeBit3 := FALSE;
   STATUS[386].EXT.BIT19 := FALSE;
   STATUS[386].EXT.BIT20 := FALSE;
   STATUS[386].EXT.AlarmSuppressed := FALSE;
   STATUS[386].EXT.AlarmPresent := FALSE;
   STATUS[386].EXT.AlarmFailUnAck := FALSE;
   STATUS[386].Status := 0;
   STATUS[386].TimeStamp := 16#0000;
   STATUS[387].EXT.AlarmWarnUnAck := FALSE;
   STATUS[387].EXT.AckRequired := FALSE;
   STATUS[387].EXT.Maintanence := FALSE;
   STATUS[387].EXT.Operation := FALSE;
   STATUS[387].EXT.Forced := FALSE;
   STATUS[387].EXT.BIT29 := FALSE;
   STATUS[387].EXT.BIT30 := FALSE;
   STATUS[387].EXT.BIT31 := FALSE;
   STATUS[387].EXT.ModeBit1 := FALSE;
   STATUS[387].EXT.ModeBit2 := FALSE;
   STATUS[387].EXT.ModeBit3 := FALSE;
   STATUS[387].EXT.BIT19 := FALSE;
   STATUS[387].EXT.BIT20 := FALSE;
   STATUS[387].EXT.AlarmSuppressed := FALSE;
   STATUS[387].EXT.AlarmPresent := FALSE;
   STATUS[387].EXT.AlarmFailUnAck := FALSE;
   STATUS[387].Status := 0;
   STATUS[387].TimeStamp := 16#0000;
   STATUS[388].EXT.AlarmWarnUnAck := FALSE;
   STATUS[388].EXT.AckRequired := FALSE;
   STATUS[388].EXT.Maintanence := FALSE;
   STATUS[388].EXT.Operation := FALSE;
   STATUS[388].EXT.Forced := FALSE;
   STATUS[388].EXT.BIT29 := FALSE;
   STATUS[388].EXT.BIT30 := FALSE;
   STATUS[388].EXT.BIT31 := FALSE;
   STATUS[388].EXT.ModeBit1 := FALSE;
   STATUS[388].EXT.ModeBit2 := FALSE;
   STATUS[388].EXT.ModeBit3 := FALSE;
   STATUS[388].EXT.BIT19 := FALSE;
   STATUS[388].EXT.BIT20 := FALSE;
   STATUS[388].EXT.AlarmSuppressed := FALSE;
   STATUS[388].EXT.AlarmPresent := FALSE;
   STATUS[388].EXT.AlarmFailUnAck := FALSE;
   STATUS[388].Status := 0;
   STATUS[388].TimeStamp := 16#0000;
   STATUS[389].EXT.AlarmWarnUnAck := FALSE;
   STATUS[389].EXT.AckRequired := FALSE;
   STATUS[389].EXT.Maintanence := FALSE;
   STATUS[389].EXT.Operation := FALSE;
   STATUS[389].EXT.Forced := FALSE;
   STATUS[389].EXT.BIT29 := FALSE;
   STATUS[389].EXT.BIT30 := FALSE;
   STATUS[389].EXT.BIT31 := FALSE;
   STATUS[389].EXT.ModeBit1 := FALSE;
   STATUS[389].EXT.ModeBit2 := FALSE;
   STATUS[389].EXT.ModeBit3 := FALSE;
   STATUS[389].EXT.BIT19 := FALSE;
   STATUS[389].EXT.BIT20 := FALSE;
   STATUS[389].EXT.AlarmSuppressed := FALSE;
   STATUS[389].EXT.AlarmPresent := FALSE;
   STATUS[389].EXT.AlarmFailUnAck := FALSE;
   STATUS[389].Status := 0;
   STATUS[389].TimeStamp := 16#0000;
   STATUS[390].EXT.AlarmWarnUnAck := FALSE;
   STATUS[390].EXT.AckRequired := FALSE;
   STATUS[390].EXT.Maintanence := FALSE;
   STATUS[390].EXT.Operation := FALSE;
   STATUS[390].EXT.Forced := FALSE;
   STATUS[390].EXT.BIT29 := FALSE;
   STATUS[390].EXT.BIT30 := FALSE;
   STATUS[390].EXT.BIT31 := FALSE;
   STATUS[390].EXT.ModeBit1 := FALSE;
   STATUS[390].EXT.ModeBit2 := FALSE;
   STATUS[390].EXT.ModeBit3 := FALSE;
   STATUS[390].EXT.BIT19 := FALSE;
   STATUS[390].EXT.BIT20 := FALSE;
   STATUS[390].EXT.AlarmSuppressed := FALSE;
   STATUS[390].EXT.AlarmPresent := FALSE;
   STATUS[390].EXT.AlarmFailUnAck := FALSE;
   STATUS[390].Status := 0;
   STATUS[390].TimeStamp := 16#0000;
   STATUS[391].EXT.AlarmWarnUnAck := FALSE;
   STATUS[391].EXT.AckRequired := FALSE;
   STATUS[391].EXT.Maintanence := FALSE;
   STATUS[391].EXT.Operation := FALSE;
   STATUS[391].EXT.Forced := FALSE;
   STATUS[391].EXT.BIT29 := FALSE;
   STATUS[391].EXT.BIT30 := FALSE;
   STATUS[391].EXT.BIT31 := FALSE;
   STATUS[391].EXT.ModeBit1 := FALSE;
   STATUS[391].EXT.ModeBit2 := FALSE;
   STATUS[391].EXT.ModeBit3 := FALSE;
   STATUS[391].EXT.BIT19 := FALSE;
   STATUS[391].EXT.BIT20 := FALSE;
   STATUS[391].EXT.AlarmSuppressed := FALSE;
   STATUS[391].EXT.AlarmPresent := FALSE;
   STATUS[391].EXT.AlarmFailUnAck := FALSE;
   STATUS[391].Status := 0;
   STATUS[391].TimeStamp := 16#0000;
   STATUS[392].EXT.AlarmWarnUnAck := FALSE;
   STATUS[392].EXT.AckRequired := FALSE;
   STATUS[392].EXT.Maintanence := FALSE;
   STATUS[392].EXT.Operation := FALSE;
   STATUS[392].EXT.Forced := FALSE;
   STATUS[392].EXT.BIT29 := FALSE;
   STATUS[392].EXT.BIT30 := FALSE;
   STATUS[392].EXT.BIT31 := FALSE;
   STATUS[392].EXT.ModeBit1 := FALSE;
   STATUS[392].EXT.ModeBit2 := FALSE;
   STATUS[392].EXT.ModeBit3 := FALSE;
   STATUS[392].EXT.BIT19 := FALSE;
   STATUS[392].EXT.BIT20 := FALSE;
   STATUS[392].EXT.AlarmSuppressed := FALSE;
   STATUS[392].EXT.AlarmPresent := FALSE;
   STATUS[392].EXT.AlarmFailUnAck := FALSE;
   STATUS[392].Status := 0;
   STATUS[392].TimeStamp := 16#0000;
   STATUS[393].EXT.AlarmWarnUnAck := FALSE;
   STATUS[393].EXT.AckRequired := FALSE;
   STATUS[393].EXT.Maintanence := FALSE;
   STATUS[393].EXT.Operation := FALSE;
   STATUS[393].EXT.Forced := FALSE;
   STATUS[393].EXT.BIT29 := FALSE;
   STATUS[393].EXT.BIT30 := FALSE;
   STATUS[393].EXT.BIT31 := FALSE;
   STATUS[393].EXT.ModeBit1 := FALSE;
   STATUS[393].EXT.ModeBit2 := FALSE;
   STATUS[393].EXT.ModeBit3 := FALSE;
   STATUS[393].EXT.BIT19 := FALSE;
   STATUS[393].EXT.BIT20 := FALSE;
   STATUS[393].EXT.AlarmSuppressed := FALSE;
   STATUS[393].EXT.AlarmPresent := FALSE;
   STATUS[393].EXT.AlarmFailUnAck := FALSE;
   STATUS[393].Status := 0;
   STATUS[393].TimeStamp := 16#0000;
   STATUS[394].EXT.AlarmWarnUnAck := FALSE;
   STATUS[394].EXT.AckRequired := FALSE;
   STATUS[394].EXT.Maintanence := FALSE;
   STATUS[394].EXT.Operation := FALSE;
   STATUS[394].EXT.Forced := FALSE;
   STATUS[394].EXT.BIT29 := FALSE;
   STATUS[394].EXT.BIT30 := FALSE;
   STATUS[394].EXT.BIT31 := FALSE;
   STATUS[394].EXT.ModeBit1 := FALSE;
   STATUS[394].EXT.ModeBit2 := FALSE;
   STATUS[394].EXT.ModeBit3 := FALSE;
   STATUS[394].EXT.BIT19 := FALSE;
   STATUS[394].EXT.BIT20 := FALSE;
   STATUS[394].EXT.AlarmSuppressed := FALSE;
   STATUS[394].EXT.AlarmPresent := FALSE;
   STATUS[394].EXT.AlarmFailUnAck := FALSE;
   STATUS[394].Status := 0;
   STATUS[394].TimeStamp := 16#0000;
   STATUS[395].EXT.AlarmWarnUnAck := FALSE;
   STATUS[395].EXT.AckRequired := FALSE;
   STATUS[395].EXT.Maintanence := FALSE;
   STATUS[395].EXT.Operation := FALSE;
   STATUS[395].EXT.Forced := FALSE;
   STATUS[395].EXT.BIT29 := FALSE;
   STATUS[395].EXT.BIT30 := FALSE;
   STATUS[395].EXT.BIT31 := FALSE;
   STATUS[395].EXT.ModeBit1 := FALSE;
   STATUS[395].EXT.ModeBit2 := FALSE;
   STATUS[395].EXT.ModeBit3 := FALSE;
   STATUS[395].EXT.BIT19 := FALSE;
   STATUS[395].EXT.BIT20 := FALSE;
   STATUS[395].EXT.AlarmSuppressed := FALSE;
   STATUS[395].EXT.AlarmPresent := FALSE;
   STATUS[395].EXT.AlarmFailUnAck := FALSE;
   STATUS[395].Status := 0;
   STATUS[395].TimeStamp := 16#0000;
   STATUS[396].EXT.AlarmWarnUnAck := FALSE;
   STATUS[396].EXT.AckRequired := FALSE;
   STATUS[396].EXT.Maintanence := FALSE;
   STATUS[396].EXT.Operation := FALSE;
   STATUS[396].EXT.Forced := FALSE;
   STATUS[396].EXT.BIT29 := FALSE;
   STATUS[396].EXT.BIT30 := FALSE;
   STATUS[396].EXT.BIT31 := FALSE;
   STATUS[396].EXT.ModeBit1 := FALSE;
   STATUS[396].EXT.ModeBit2 := FALSE;
   STATUS[396].EXT.ModeBit3 := FALSE;
   STATUS[396].EXT.BIT19 := FALSE;
   STATUS[396].EXT.BIT20 := FALSE;
   STATUS[396].EXT.AlarmSuppressed := FALSE;
   STATUS[396].EXT.AlarmPresent := FALSE;
   STATUS[396].EXT.AlarmFailUnAck := FALSE;
   STATUS[396].Status := 0;
   STATUS[396].TimeStamp := 16#0000;
   STATUS[397].EXT.AlarmWarnUnAck := FALSE;
   STATUS[397].EXT.AckRequired := FALSE;
   STATUS[397].EXT.Maintanence := FALSE;
   STATUS[397].EXT.Operation := FALSE;
   STATUS[397].EXT.Forced := FALSE;
   STATUS[397].EXT.BIT29 := FALSE;
   STATUS[397].EXT.BIT30 := FALSE;
   STATUS[397].EXT.BIT31 := FALSE;
   STATUS[397].EXT.ModeBit1 := FALSE;
   STATUS[397].EXT.ModeBit2 := FALSE;
   STATUS[397].EXT.ModeBit3 := FALSE;
   STATUS[397].EXT.BIT19 := FALSE;
   STATUS[397].EXT.BIT20 := FALSE;
   STATUS[397].EXT.AlarmSuppressed := FALSE;
   STATUS[397].EXT.AlarmPresent := FALSE;
   STATUS[397].EXT.AlarmFailUnAck := FALSE;
   STATUS[397].Status := 0;
   STATUS[397].TimeStamp := 16#0000;
   STATUS[398].EXT.AlarmWarnUnAck := FALSE;
   STATUS[398].EXT.AckRequired := FALSE;
   STATUS[398].EXT.Maintanence := FALSE;
   STATUS[398].EXT.Operation := FALSE;
   STATUS[398].EXT.Forced := FALSE;
   STATUS[398].EXT.BIT29 := FALSE;
   STATUS[398].EXT.BIT30 := FALSE;
   STATUS[398].EXT.BIT31 := FALSE;
   STATUS[398].EXT.ModeBit1 := FALSE;
   STATUS[398].EXT.ModeBit2 := FALSE;
   STATUS[398].EXT.ModeBit3 := FALSE;
   STATUS[398].EXT.BIT19 := FALSE;
   STATUS[398].EXT.BIT20 := FALSE;
   STATUS[398].EXT.AlarmSuppressed := FALSE;
   STATUS[398].EXT.AlarmPresent := FALSE;
   STATUS[398].EXT.AlarmFailUnAck := FALSE;
   STATUS[398].Status := 0;
   STATUS[398].TimeStamp := 16#0000;
   STATUS[399].EXT.AlarmWarnUnAck := FALSE;
   STATUS[399].EXT.AckRequired := FALSE;
   STATUS[399].EXT.Maintanence := FALSE;
   STATUS[399].EXT.Operation := FALSE;
   STATUS[399].EXT.Forced := FALSE;
   STATUS[399].EXT.BIT29 := FALSE;
   STATUS[399].EXT.BIT30 := FALSE;
   STATUS[399].EXT.BIT31 := FALSE;
   STATUS[399].EXT.ModeBit1 := FALSE;
   STATUS[399].EXT.ModeBit2 := FALSE;
   STATUS[399].EXT.ModeBit3 := FALSE;
   STATUS[399].EXT.BIT19 := FALSE;
   STATUS[399].EXT.BIT20 := FALSE;
   STATUS[399].EXT.AlarmSuppressed := FALSE;
   STATUS[399].EXT.AlarmPresent := FALSE;
   STATUS[399].EXT.AlarmFailUnAck := FALSE;
   STATUS[399].Status := 0;
   STATUS[399].TimeStamp := 16#0000;
   STATUS[400].EXT.AlarmWarnUnAck := FALSE;
   STATUS[400].EXT.AckRequired := FALSE;
   STATUS[400].EXT.Maintanence := FALSE;
   STATUS[400].EXT.Operation := FALSE;
   STATUS[400].EXT.Forced := FALSE;
   STATUS[400].EXT.BIT29 := FALSE;
   STATUS[400].EXT.BIT30 := FALSE;
   STATUS[400].EXT.BIT31 := FALSE;
   STATUS[400].EXT.ModeBit1 := FALSE;
   STATUS[400].EXT.ModeBit2 := FALSE;
   STATUS[400].EXT.ModeBit3 := FALSE;
   STATUS[400].EXT.BIT19 := FALSE;
   STATUS[400].EXT.BIT20 := FALSE;
   STATUS[400].EXT.AlarmSuppressed := FALSE;
   STATUS[400].EXT.AlarmPresent := FALSE;
   STATUS[400].EXT.AlarmFailUnAck := FALSE;
   STATUS[400].Status := 0;
   STATUS[400].TimeStamp := 16#0000;
   STATUS[401].EXT.AlarmWarnUnAck := FALSE;
   STATUS[401].EXT.AckRequired := FALSE;
   STATUS[401].EXT.Maintanence := FALSE;
   STATUS[401].EXT.Operation := FALSE;
   STATUS[401].EXT.Forced := FALSE;
   STATUS[401].EXT.BIT29 := FALSE;
   STATUS[401].EXT.BIT30 := FALSE;
   STATUS[401].EXT.BIT31 := FALSE;
   STATUS[401].EXT.ModeBit1 := FALSE;
   STATUS[401].EXT.ModeBit2 := FALSE;
   STATUS[401].EXT.ModeBit3 := FALSE;
   STATUS[401].EXT.BIT19 := FALSE;
   STATUS[401].EXT.BIT20 := FALSE;
   STATUS[401].EXT.AlarmSuppressed := FALSE;
   STATUS[401].EXT.AlarmPresent := FALSE;
   STATUS[401].EXT.AlarmFailUnAck := FALSE;
   STATUS[401].Status := 0;
   STATUS[401].TimeStamp := 16#0000;
   STATUS[402].EXT.AlarmWarnUnAck := FALSE;
   STATUS[402].EXT.AckRequired := FALSE;
   STATUS[402].EXT.Maintanence := FALSE;
   STATUS[402].EXT.Operation := FALSE;
   STATUS[402].EXT.Forced := FALSE;
   STATUS[402].EXT.BIT29 := FALSE;
   STATUS[402].EXT.BIT30 := FALSE;
   STATUS[402].EXT.BIT31 := FALSE;
   STATUS[402].EXT.ModeBit1 := FALSE;
   STATUS[402].EXT.ModeBit2 := FALSE;
   STATUS[402].EXT.ModeBit3 := FALSE;
   STATUS[402].EXT.BIT19 := FALSE;
   STATUS[402].EXT.BIT20 := FALSE;
   STATUS[402].EXT.AlarmSuppressed := FALSE;
   STATUS[402].EXT.AlarmPresent := FALSE;
   STATUS[402].EXT.AlarmFailUnAck := FALSE;
   STATUS[402].Status := 0;
   STATUS[402].TimeStamp := 16#0000;
   STATUS[403].EXT.AlarmWarnUnAck := FALSE;
   STATUS[403].EXT.AckRequired := FALSE;
   STATUS[403].EXT.Maintanence := FALSE;
   STATUS[403].EXT.Operation := FALSE;
   STATUS[403].EXT.Forced := FALSE;
   STATUS[403].EXT.BIT29 := FALSE;
   STATUS[403].EXT.BIT30 := FALSE;
   STATUS[403].EXT.BIT31 := FALSE;
   STATUS[403].EXT.ModeBit1 := FALSE;
   STATUS[403].EXT.ModeBit2 := FALSE;
   STATUS[403].EXT.ModeBit3 := FALSE;
   STATUS[403].EXT.BIT19 := FALSE;
   STATUS[403].EXT.BIT20 := FALSE;
   STATUS[403].EXT.AlarmSuppressed := FALSE;
   STATUS[403].EXT.AlarmPresent := FALSE;
   STATUS[403].EXT.AlarmFailUnAck := FALSE;
   STATUS[403].Status := 0;
   STATUS[403].TimeStamp := 16#0000;
   STATUS[404].EXT.AlarmWarnUnAck := FALSE;
   STATUS[404].EXT.AckRequired := FALSE;
   STATUS[404].EXT.Maintanence := FALSE;
   STATUS[404].EXT.Operation := FALSE;
   STATUS[404].EXT.Forced := FALSE;
   STATUS[404].EXT.BIT29 := FALSE;
   STATUS[404].EXT.BIT30 := FALSE;
   STATUS[404].EXT.BIT31 := FALSE;
   STATUS[404].EXT.ModeBit1 := FALSE;
   STATUS[404].EXT.ModeBit2 := FALSE;
   STATUS[404].EXT.ModeBit3 := FALSE;
   STATUS[404].EXT.BIT19 := FALSE;
   STATUS[404].EXT.BIT20 := FALSE;
   STATUS[404].EXT.AlarmSuppressed := FALSE;
   STATUS[404].EXT.AlarmPresent := FALSE;
   STATUS[404].EXT.AlarmFailUnAck := FALSE;
   STATUS[404].Status := 0;
   STATUS[404].TimeStamp := 16#0000;
   STATUS[405].EXT.AlarmWarnUnAck := FALSE;
   STATUS[405].EXT.AckRequired := FALSE;
   STATUS[405].EXT.Maintanence := FALSE;
   STATUS[405].EXT.Operation := FALSE;
   STATUS[405].EXT.Forced := FALSE;
   STATUS[405].EXT.BIT29 := FALSE;
   STATUS[405].EXT.BIT30 := FALSE;
   STATUS[405].EXT.BIT31 := FALSE;
   STATUS[405].EXT.ModeBit1 := FALSE;
   STATUS[405].EXT.ModeBit2 := FALSE;
   STATUS[405].EXT.ModeBit3 := FALSE;
   STATUS[405].EXT.BIT19 := FALSE;
   STATUS[405].EXT.BIT20 := FALSE;
   STATUS[405].EXT.AlarmSuppressed := FALSE;
   STATUS[405].EXT.AlarmPresent := FALSE;
   STATUS[405].EXT.AlarmFailUnAck := FALSE;
   STATUS[405].Status := 0;
   STATUS[405].TimeStamp := 16#0000;
   STATUS[406].EXT.AlarmWarnUnAck := FALSE;
   STATUS[406].EXT.AckRequired := FALSE;
   STATUS[406].EXT.Maintanence := FALSE;
   STATUS[406].EXT.Operation := FALSE;
   STATUS[406].EXT.Forced := FALSE;
   STATUS[406].EXT.BIT29 := FALSE;
   STATUS[406].EXT.BIT30 := FALSE;
   STATUS[406].EXT.BIT31 := FALSE;
   STATUS[406].EXT.ModeBit1 := FALSE;
   STATUS[406].EXT.ModeBit2 := FALSE;
   STATUS[406].EXT.ModeBit3 := FALSE;
   STATUS[406].EXT.BIT19 := FALSE;
   STATUS[406].EXT.BIT20 := FALSE;
   STATUS[406].EXT.AlarmSuppressed := FALSE;
   STATUS[406].EXT.AlarmPresent := FALSE;
   STATUS[406].EXT.AlarmFailUnAck := FALSE;
   STATUS[406].Status := 0;
   STATUS[406].TimeStamp := 16#0000;
   STATUS[407].EXT.AlarmWarnUnAck := FALSE;
   STATUS[407].EXT.AckRequired := FALSE;
   STATUS[407].EXT.Maintanence := FALSE;
   STATUS[407].EXT.Operation := FALSE;
   STATUS[407].EXT.Forced := FALSE;
   STATUS[407].EXT.BIT29 := FALSE;
   STATUS[407].EXT.BIT30 := FALSE;
   STATUS[407].EXT.BIT31 := FALSE;
   STATUS[407].EXT.ModeBit1 := FALSE;
   STATUS[407].EXT.ModeBit2 := FALSE;
   STATUS[407].EXT.ModeBit3 := FALSE;
   STATUS[407].EXT.BIT19 := FALSE;
   STATUS[407].EXT.BIT20 := FALSE;
   STATUS[407].EXT.AlarmSuppressed := FALSE;
   STATUS[407].EXT.AlarmPresent := FALSE;
   STATUS[407].EXT.AlarmFailUnAck := FALSE;
   STATUS[407].Status := 0;
   STATUS[407].TimeStamp := 16#0000;
   STATUS[408].EXT.AlarmWarnUnAck := FALSE;
   STATUS[408].EXT.AckRequired := FALSE;
   STATUS[408].EXT.Maintanence := FALSE;
   STATUS[408].EXT.Operation := FALSE;
   STATUS[408].EXT.Forced := FALSE;
   STATUS[408].EXT.BIT29 := FALSE;
   STATUS[408].EXT.BIT30 := FALSE;
   STATUS[408].EXT.BIT31 := FALSE;
   STATUS[408].EXT.ModeBit1 := FALSE;
   STATUS[408].EXT.ModeBit2 := FALSE;
   STATUS[408].EXT.ModeBit3 := FALSE;
   STATUS[408].EXT.BIT19 := FALSE;
   STATUS[408].EXT.BIT20 := FALSE;
   STATUS[408].EXT.AlarmSuppressed := FALSE;
   STATUS[408].EXT.AlarmPresent := FALSE;
   STATUS[408].EXT.AlarmFailUnAck := FALSE;
   STATUS[408].Status := 0;
   STATUS[408].TimeStamp := 16#0000;
   STATUS[409].EXT.AlarmWarnUnAck := FALSE;
   STATUS[409].EXT.AckRequired := FALSE;
   STATUS[409].EXT.Maintanence := FALSE;
   STATUS[409].EXT.Operation := FALSE;
   STATUS[409].EXT.Forced := FALSE;
   STATUS[409].EXT.BIT29 := FALSE;
   STATUS[409].EXT.BIT30 := FALSE;
   STATUS[409].EXT.BIT31 := FALSE;
   STATUS[409].EXT.ModeBit1 := FALSE;
   STATUS[409].EXT.ModeBit2 := FALSE;
   STATUS[409].EXT.ModeBit3 := FALSE;
   STATUS[409].EXT.BIT19 := FALSE;
   STATUS[409].EXT.BIT20 := FALSE;
   STATUS[409].EXT.AlarmSuppressed := FALSE;
   STATUS[409].EXT.AlarmPresent := FALSE;
   STATUS[409].EXT.AlarmFailUnAck := FALSE;
   STATUS[409].Status := 0;
   STATUS[409].TimeStamp := 16#0000;
   STATUS[410].EXT.AlarmWarnUnAck := FALSE;
   STATUS[410].EXT.AckRequired := FALSE;
   STATUS[410].EXT.Maintanence := FALSE;
   STATUS[410].EXT.Operation := FALSE;
   STATUS[410].EXT.Forced := FALSE;
   STATUS[410].EXT.BIT29 := FALSE;
   STATUS[410].EXT.BIT30 := FALSE;
   STATUS[410].EXT.BIT31 := FALSE;
   STATUS[410].EXT.ModeBit1 := FALSE;
   STATUS[410].EXT.ModeBit2 := FALSE;
   STATUS[410].EXT.ModeBit3 := FALSE;
   STATUS[410].EXT.BIT19 := FALSE;
   STATUS[410].EXT.BIT20 := FALSE;
   STATUS[410].EXT.AlarmSuppressed := FALSE;
   STATUS[410].EXT.AlarmPresent := FALSE;
   STATUS[410].EXT.AlarmFailUnAck := FALSE;
   STATUS[410].Status := 0;
   STATUS[410].TimeStamp := 16#0000;
   STATUS[411].EXT.AlarmWarnUnAck := FALSE;
   STATUS[411].EXT.AckRequired := FALSE;
   STATUS[411].EXT.Maintanence := FALSE;
   STATUS[411].EXT.Operation := FALSE;
   STATUS[411].EXT.Forced := FALSE;
   STATUS[411].EXT.BIT29 := FALSE;
   STATUS[411].EXT.BIT30 := FALSE;
   STATUS[411].EXT.BIT31 := FALSE;
   STATUS[411].EXT.ModeBit1 := FALSE;
   STATUS[411].EXT.ModeBit2 := FALSE;
   STATUS[411].EXT.ModeBit3 := FALSE;
   STATUS[411].EXT.BIT19 := FALSE;
   STATUS[411].EXT.BIT20 := FALSE;
   STATUS[411].EXT.AlarmSuppressed := FALSE;
   STATUS[411].EXT.AlarmPresent := FALSE;
   STATUS[411].EXT.AlarmFailUnAck := FALSE;
   STATUS[411].Status := 0;
   STATUS[411].TimeStamp := 16#0000;
   STATUS[412].EXT.AlarmWarnUnAck := FALSE;
   STATUS[412].EXT.AckRequired := FALSE;
   STATUS[412].EXT.Maintanence := FALSE;
   STATUS[412].EXT.Operation := FALSE;
   STATUS[412].EXT.Forced := FALSE;
   STATUS[412].EXT.BIT29 := FALSE;
   STATUS[412].EXT.BIT30 := FALSE;
   STATUS[412].EXT.BIT31 := FALSE;
   STATUS[412].EXT.ModeBit1 := FALSE;
   STATUS[412].EXT.ModeBit2 := FALSE;
   STATUS[412].EXT.ModeBit3 := FALSE;
   STATUS[412].EXT.BIT19 := FALSE;
   STATUS[412].EXT.BIT20 := FALSE;
   STATUS[412].EXT.AlarmSuppressed := FALSE;
   STATUS[412].EXT.AlarmPresent := FALSE;
   STATUS[412].EXT.AlarmFailUnAck := FALSE;
   STATUS[412].Status := 0;
   STATUS[412].TimeStamp := 16#0000;
   STATUS[413].EXT.AlarmWarnUnAck := FALSE;
   STATUS[413].EXT.AckRequired := FALSE;
   STATUS[413].EXT.Maintanence := FALSE;
   STATUS[413].EXT.Operation := FALSE;
   STATUS[413].EXT.Forced := FALSE;
   STATUS[413].EXT.BIT29 := FALSE;
   STATUS[413].EXT.BIT30 := FALSE;
   STATUS[413].EXT.BIT31 := FALSE;
   STATUS[413].EXT.ModeBit1 := FALSE;
   STATUS[413].EXT.ModeBit2 := FALSE;
   STATUS[413].EXT.ModeBit3 := FALSE;
   STATUS[413].EXT.BIT19 := FALSE;
   STATUS[413].EXT.BIT20 := FALSE;
   STATUS[413].EXT.AlarmSuppressed := FALSE;
   STATUS[413].EXT.AlarmPresent := FALSE;
   STATUS[413].EXT.AlarmFailUnAck := FALSE;
   STATUS[413].Status := 0;
   STATUS[413].TimeStamp := 16#0000;
   STATUS[414].EXT.AlarmWarnUnAck := FALSE;
   STATUS[414].EXT.AckRequired := FALSE;
   STATUS[414].EXT.Maintanence := FALSE;
   STATUS[414].EXT.Operation := FALSE;
   STATUS[414].EXT.Forced := FALSE;
   STATUS[414].EXT.BIT29 := FALSE;
   STATUS[414].EXT.BIT30 := FALSE;
   STATUS[414].EXT.BIT31 := FALSE;
   STATUS[414].EXT.ModeBit1 := FALSE;
   STATUS[414].EXT.ModeBit2 := FALSE;
   STATUS[414].EXT.ModeBit3 := FALSE;
   STATUS[414].EXT.BIT19 := FALSE;
   STATUS[414].EXT.BIT20 := FALSE;
   STATUS[414].EXT.AlarmSuppressed := FALSE;
   STATUS[414].EXT.AlarmPresent := FALSE;
   STATUS[414].EXT.AlarmFailUnAck := FALSE;
   STATUS[414].Status := 0;
   STATUS[414].TimeStamp := 16#0000;
   STATUS[415].EXT.AlarmWarnUnAck := FALSE;
   STATUS[415].EXT.AckRequired := FALSE;
   STATUS[415].EXT.Maintanence := FALSE;
   STATUS[415].EXT.Operation := FALSE;
   STATUS[415].EXT.Forced := FALSE;
   STATUS[415].EXT.BIT29 := FALSE;
   STATUS[415].EXT.BIT30 := FALSE;
   STATUS[415].EXT.BIT31 := FALSE;
   STATUS[415].EXT.ModeBit1 := FALSE;
   STATUS[415].EXT.ModeBit2 := FALSE;
   STATUS[415].EXT.ModeBit3 := FALSE;
   STATUS[415].EXT.BIT19 := FALSE;
   STATUS[415].EXT.BIT20 := FALSE;
   STATUS[415].EXT.AlarmSuppressed := FALSE;
   STATUS[415].EXT.AlarmPresent := FALSE;
   STATUS[415].EXT.AlarmFailUnAck := FALSE;
   STATUS[415].Status := 0;
   STATUS[415].TimeStamp := 16#0000;
   STATUS[416].EXT.AlarmWarnUnAck := FALSE;
   STATUS[416].EXT.AckRequired := FALSE;
   STATUS[416].EXT.Maintanence := FALSE;
   STATUS[416].EXT.Operation := FALSE;
   STATUS[416].EXT.Forced := FALSE;
   STATUS[416].EXT.BIT29 := FALSE;
   STATUS[416].EXT.BIT30 := FALSE;
   STATUS[416].EXT.BIT31 := FALSE;
   STATUS[416].EXT.ModeBit1 := FALSE;
   STATUS[416].EXT.ModeBit2 := FALSE;
   STATUS[416].EXT.ModeBit3 := FALSE;
   STATUS[416].EXT.BIT19 := FALSE;
   STATUS[416].EXT.BIT20 := FALSE;
   STATUS[416].EXT.AlarmSuppressed := FALSE;
   STATUS[416].EXT.AlarmPresent := FALSE;
   STATUS[416].EXT.AlarmFailUnAck := FALSE;
   STATUS[416].Status := 0;
   STATUS[416].TimeStamp := 16#0000;
   STATUS[417].EXT.AlarmWarnUnAck := FALSE;
   STATUS[417].EXT.AckRequired := FALSE;
   STATUS[417].EXT.Maintanence := FALSE;
   STATUS[417].EXT.Operation := FALSE;
   STATUS[417].EXT.Forced := FALSE;
   STATUS[417].EXT.BIT29 := FALSE;
   STATUS[417].EXT.BIT30 := FALSE;
   STATUS[417].EXT.BIT31 := FALSE;
   STATUS[417].EXT.ModeBit1 := FALSE;
   STATUS[417].EXT.ModeBit2 := FALSE;
   STATUS[417].EXT.ModeBit3 := FALSE;
   STATUS[417].EXT.BIT19 := FALSE;
   STATUS[417].EXT.BIT20 := FALSE;
   STATUS[417].EXT.AlarmSuppressed := FALSE;
   STATUS[417].EXT.AlarmPresent := FALSE;
   STATUS[417].EXT.AlarmFailUnAck := FALSE;
   STATUS[417].Status := 0;
   STATUS[417].TimeStamp := 16#0000;
   STATUS[418].EXT.AlarmWarnUnAck := FALSE;
   STATUS[418].EXT.AckRequired := FALSE;
   STATUS[418].EXT.Maintanence := FALSE;
   STATUS[418].EXT.Operation := FALSE;
   STATUS[418].EXT.Forced := FALSE;
   STATUS[418].EXT.BIT29 := FALSE;
   STATUS[418].EXT.BIT30 := FALSE;
   STATUS[418].EXT.BIT31 := FALSE;
   STATUS[418].EXT.ModeBit1 := FALSE;
   STATUS[418].EXT.ModeBit2 := FALSE;
   STATUS[418].EXT.ModeBit3 := FALSE;
   STATUS[418].EXT.BIT19 := FALSE;
   STATUS[418].EXT.BIT20 := FALSE;
   STATUS[418].EXT.AlarmSuppressed := FALSE;
   STATUS[418].EXT.AlarmPresent := FALSE;
   STATUS[418].EXT.AlarmFailUnAck := FALSE;
   STATUS[418].Status := 0;
   STATUS[418].TimeStamp := 16#0000;
   STATUS[419].EXT.AlarmWarnUnAck := FALSE;
   STATUS[419].EXT.AckRequired := FALSE;
   STATUS[419].EXT.Maintanence := FALSE;
   STATUS[419].EXT.Operation := FALSE;
   STATUS[419].EXT.Forced := FALSE;
   STATUS[419].EXT.BIT29 := FALSE;
   STATUS[419].EXT.BIT30 := FALSE;
   STATUS[419].EXT.BIT31 := FALSE;
   STATUS[419].EXT.ModeBit1 := FALSE;
   STATUS[419].EXT.ModeBit2 := FALSE;
   STATUS[419].EXT.ModeBit3 := FALSE;
   STATUS[419].EXT.BIT19 := FALSE;
   STATUS[419].EXT.BIT20 := FALSE;
   STATUS[419].EXT.AlarmSuppressed := FALSE;
   STATUS[419].EXT.AlarmPresent := FALSE;
   STATUS[419].EXT.AlarmFailUnAck := FALSE;
   STATUS[419].Status := 0;
   STATUS[419].TimeStamp := 16#0000;
   STATUS[420].EXT.AlarmWarnUnAck := FALSE;
   STATUS[420].EXT.AckRequired := FALSE;
   STATUS[420].EXT.Maintanence := FALSE;
   STATUS[420].EXT.Operation := FALSE;
   STATUS[420].EXT.Forced := FALSE;
   STATUS[420].EXT.BIT29 := FALSE;
   STATUS[420].EXT.BIT30 := FALSE;
   STATUS[420].EXT.BIT31 := FALSE;
   STATUS[420].EXT.ModeBit1 := FALSE;
   STATUS[420].EXT.ModeBit2 := FALSE;
   STATUS[420].EXT.ModeBit3 := FALSE;
   STATUS[420].EXT.BIT19 := FALSE;
   STATUS[420].EXT.BIT20 := FALSE;
   STATUS[420].EXT.AlarmSuppressed := FALSE;
   STATUS[420].EXT.AlarmPresent := FALSE;
   STATUS[420].EXT.AlarmFailUnAck := FALSE;
   STATUS[420].Status := 0;
   STATUS[420].TimeStamp := 16#0000;
   STATUS[421].EXT.AlarmWarnUnAck := FALSE;
   STATUS[421].EXT.AckRequired := FALSE;
   STATUS[421].EXT.Maintanence := FALSE;
   STATUS[421].EXT.Operation := FALSE;
   STATUS[421].EXT.Forced := FALSE;
   STATUS[421].EXT.BIT29 := FALSE;
   STATUS[421].EXT.BIT30 := FALSE;
   STATUS[421].EXT.BIT31 := FALSE;
   STATUS[421].EXT.ModeBit1 := FALSE;
   STATUS[421].EXT.ModeBit2 := FALSE;
   STATUS[421].EXT.ModeBit3 := FALSE;
   STATUS[421].EXT.BIT19 := FALSE;
   STATUS[421].EXT.BIT20 := FALSE;
   STATUS[421].EXT.AlarmSuppressed := FALSE;
   STATUS[421].EXT.AlarmPresent := FALSE;
   STATUS[421].EXT.AlarmFailUnAck := FALSE;
   STATUS[421].Status := 0;
   STATUS[421].TimeStamp := 16#0000;
   STATUS[422].EXT.AlarmWarnUnAck := FALSE;
   STATUS[422].EXT.AckRequired := FALSE;
   STATUS[422].EXT.Maintanence := FALSE;
   STATUS[422].EXT.Operation := FALSE;
   STATUS[422].EXT.Forced := FALSE;
   STATUS[422].EXT.BIT29 := FALSE;
   STATUS[422].EXT.BIT30 := FALSE;
   STATUS[422].EXT.BIT31 := FALSE;
   STATUS[422].EXT.ModeBit1 := FALSE;
   STATUS[422].EXT.ModeBit2 := FALSE;
   STATUS[422].EXT.ModeBit3 := FALSE;
   STATUS[422].EXT.BIT19 := FALSE;
   STATUS[422].EXT.BIT20 := FALSE;
   STATUS[422].EXT.AlarmSuppressed := FALSE;
   STATUS[422].EXT.AlarmPresent := FALSE;
   STATUS[422].EXT.AlarmFailUnAck := FALSE;
   STATUS[422].Status := 0;
   STATUS[422].TimeStamp := 16#0000;
   STATUS[423].EXT.AlarmWarnUnAck := FALSE;
   STATUS[423].EXT.AckRequired := FALSE;
   STATUS[423].EXT.Maintanence := FALSE;
   STATUS[423].EXT.Operation := FALSE;
   STATUS[423].EXT.Forced := FALSE;
   STATUS[423].EXT.BIT29 := FALSE;
   STATUS[423].EXT.BIT30 := FALSE;
   STATUS[423].EXT.BIT31 := FALSE;
   STATUS[423].EXT.ModeBit1 := FALSE;
   STATUS[423].EXT.ModeBit2 := FALSE;
   STATUS[423].EXT.ModeBit3 := FALSE;
   STATUS[423].EXT.BIT19 := FALSE;
   STATUS[423].EXT.BIT20 := FALSE;
   STATUS[423].EXT.AlarmSuppressed := FALSE;
   STATUS[423].EXT.AlarmPresent := FALSE;
   STATUS[423].EXT.AlarmFailUnAck := FALSE;
   STATUS[423].Status := 0;
   STATUS[423].TimeStamp := 16#0000;
   STATUS[424].EXT.AlarmWarnUnAck := FALSE;
   STATUS[424].EXT.AckRequired := FALSE;
   STATUS[424].EXT.Maintanence := FALSE;
   STATUS[424].EXT.Operation := FALSE;
   STATUS[424].EXT.Forced := FALSE;
   STATUS[424].EXT.BIT29 := FALSE;
   STATUS[424].EXT.BIT30 := FALSE;
   STATUS[424].EXT.BIT31 := FALSE;
   STATUS[424].EXT.ModeBit1 := FALSE;
   STATUS[424].EXT.ModeBit2 := FALSE;
   STATUS[424].EXT.ModeBit3 := FALSE;
   STATUS[424].EXT.BIT19 := FALSE;
   STATUS[424].EXT.BIT20 := FALSE;
   STATUS[424].EXT.AlarmSuppressed := FALSE;
   STATUS[424].EXT.AlarmPresent := FALSE;
   STATUS[424].EXT.AlarmFailUnAck := FALSE;
   STATUS[424].Status := 0;
   STATUS[424].TimeStamp := 16#0000;
   STATUS[425].EXT.AlarmWarnUnAck := FALSE;
   STATUS[425].EXT.AckRequired := FALSE;
   STATUS[425].EXT.Maintanence := FALSE;
   STATUS[425].EXT.Operation := FALSE;
   STATUS[425].EXT.Forced := FALSE;
   STATUS[425].EXT.BIT29 := FALSE;
   STATUS[425].EXT.BIT30 := FALSE;
   STATUS[425].EXT.BIT31 := FALSE;
   STATUS[425].EXT.ModeBit1 := FALSE;
   STATUS[425].EXT.ModeBit2 := FALSE;
   STATUS[425].EXT.ModeBit3 := FALSE;
   STATUS[425].EXT.BIT19 := FALSE;
   STATUS[425].EXT.BIT20 := FALSE;
   STATUS[425].EXT.AlarmSuppressed := FALSE;
   STATUS[425].EXT.AlarmPresent := FALSE;
   STATUS[425].EXT.AlarmFailUnAck := FALSE;
   STATUS[425].Status := 0;
   STATUS[425].TimeStamp := 16#0000;
   STATUS[426].EXT.AlarmWarnUnAck := FALSE;
   STATUS[426].EXT.AckRequired := FALSE;
   STATUS[426].EXT.Maintanence := FALSE;
   STATUS[426].EXT.Operation := FALSE;
   STATUS[426].EXT.Forced := FALSE;
   STATUS[426].EXT.BIT29 := FALSE;
   STATUS[426].EXT.BIT30 := FALSE;
   STATUS[426].EXT.BIT31 := FALSE;
   STATUS[426].EXT.ModeBit1 := FALSE;
   STATUS[426].EXT.ModeBit2 := FALSE;
   STATUS[426].EXT.ModeBit3 := FALSE;
   STATUS[426].EXT.BIT19 := FALSE;
   STATUS[426].EXT.BIT20 := FALSE;
   STATUS[426].EXT.AlarmSuppressed := FALSE;
   STATUS[426].EXT.AlarmPresent := FALSE;
   STATUS[426].EXT.AlarmFailUnAck := FALSE;
   STATUS[426].Status := 0;
   STATUS[426].TimeStamp := 16#0000;
   STATUS[427].EXT.AlarmWarnUnAck := FALSE;
   STATUS[427].EXT.AckRequired := FALSE;
   STATUS[427].EXT.Maintanence := FALSE;
   STATUS[427].EXT.Operation := FALSE;
   STATUS[427].EXT.Forced := FALSE;
   STATUS[427].EXT.BIT29 := FALSE;
   STATUS[427].EXT.BIT30 := FALSE;
   STATUS[427].EXT.BIT31 := FALSE;
   STATUS[427].EXT.ModeBit1 := FALSE;
   STATUS[427].EXT.ModeBit2 := FALSE;
   STATUS[427].EXT.ModeBit3 := FALSE;
   STATUS[427].EXT.BIT19 := FALSE;
   STATUS[427].EXT.BIT20 := FALSE;
   STATUS[427].EXT.AlarmSuppressed := FALSE;
   STATUS[427].EXT.AlarmPresent := FALSE;
   STATUS[427].EXT.AlarmFailUnAck := FALSE;
   STATUS[427].Status := 0;
   STATUS[427].TimeStamp := 16#0000;
   STATUS[428].EXT.AlarmWarnUnAck := FALSE;
   STATUS[428].EXT.AckRequired := FALSE;
   STATUS[428].EXT.Maintanence := FALSE;
   STATUS[428].EXT.Operation := FALSE;
   STATUS[428].EXT.Forced := FALSE;
   STATUS[428].EXT.BIT29 := FALSE;
   STATUS[428].EXT.BIT30 := FALSE;
   STATUS[428].EXT.BIT31 := FALSE;
   STATUS[428].EXT.ModeBit1 := FALSE;
   STATUS[428].EXT.ModeBit2 := FALSE;
   STATUS[428].EXT.ModeBit3 := FALSE;
   STATUS[428].EXT.BIT19 := FALSE;
   STATUS[428].EXT.BIT20 := FALSE;
   STATUS[428].EXT.AlarmSuppressed := FALSE;
   STATUS[428].EXT.AlarmPresent := FALSE;
   STATUS[428].EXT.AlarmFailUnAck := FALSE;
   STATUS[428].Status := 0;
   STATUS[428].TimeStamp := 16#0000;
   STATUS[429].EXT.AlarmWarnUnAck := FALSE;
   STATUS[429].EXT.AckRequired := FALSE;
   STATUS[429].EXT.Maintanence := FALSE;
   STATUS[429].EXT.Operation := FALSE;
   STATUS[429].EXT.Forced := FALSE;
   STATUS[429].EXT.BIT29 := FALSE;
   STATUS[429].EXT.BIT30 := FALSE;
   STATUS[429].EXT.BIT31 := FALSE;
   STATUS[429].EXT.ModeBit1 := FALSE;
   STATUS[429].EXT.ModeBit2 := FALSE;
   STATUS[429].EXT.ModeBit3 := FALSE;
   STATUS[429].EXT.BIT19 := FALSE;
   STATUS[429].EXT.BIT20 := FALSE;
   STATUS[429].EXT.AlarmSuppressed := FALSE;
   STATUS[429].EXT.AlarmPresent := FALSE;
   STATUS[429].EXT.AlarmFailUnAck := FALSE;
   STATUS[429].Status := 0;
   STATUS[429].TimeStamp := 16#0000;
   STATUS[430].EXT.AlarmWarnUnAck := FALSE;
   STATUS[430].EXT.AckRequired := FALSE;
   STATUS[430].EXT.Maintanence := FALSE;
   STATUS[430].EXT.Operation := FALSE;
   STATUS[430].EXT.Forced := FALSE;
   STATUS[430].EXT.BIT29 := FALSE;
   STATUS[430].EXT.BIT30 := FALSE;
   STATUS[430].EXT.BIT31 := FALSE;
   STATUS[430].EXT.ModeBit1 := FALSE;
   STATUS[430].EXT.ModeBit2 := FALSE;
   STATUS[430].EXT.ModeBit3 := FALSE;
   STATUS[430].EXT.BIT19 := FALSE;
   STATUS[430].EXT.BIT20 := FALSE;
   STATUS[430].EXT.AlarmSuppressed := FALSE;
   STATUS[430].EXT.AlarmPresent := FALSE;
   STATUS[430].EXT.AlarmFailUnAck := FALSE;
   STATUS[430].Status := 0;
   STATUS[430].TimeStamp := 16#0000;
   STATUS[431].EXT.AlarmWarnUnAck := FALSE;
   STATUS[431].EXT.AckRequired := FALSE;
   STATUS[431].EXT.Maintanence := FALSE;
   STATUS[431].EXT.Operation := FALSE;
   STATUS[431].EXT.Forced := FALSE;
   STATUS[431].EXT.BIT29 := FALSE;
   STATUS[431].EXT.BIT30 := FALSE;
   STATUS[431].EXT.BIT31 := FALSE;
   STATUS[431].EXT.ModeBit1 := FALSE;
   STATUS[431].EXT.ModeBit2 := FALSE;
   STATUS[431].EXT.ModeBit3 := FALSE;
   STATUS[431].EXT.BIT19 := FALSE;
   STATUS[431].EXT.BIT20 := FALSE;
   STATUS[431].EXT.AlarmSuppressed := FALSE;
   STATUS[431].EXT.AlarmPresent := FALSE;
   STATUS[431].EXT.AlarmFailUnAck := FALSE;
   STATUS[431].Status := 0;
   STATUS[431].TimeStamp := 16#0000;
   STATUS[432].EXT.AlarmWarnUnAck := FALSE;
   STATUS[432].EXT.AckRequired := FALSE;
   STATUS[432].EXT.Maintanence := FALSE;
   STATUS[432].EXT.Operation := FALSE;
   STATUS[432].EXT.Forced := FALSE;
   STATUS[432].EXT.BIT29 := FALSE;
   STATUS[432].EXT.BIT30 := FALSE;
   STATUS[432].EXT.BIT31 := FALSE;
   STATUS[432].EXT.ModeBit1 := FALSE;
   STATUS[432].EXT.ModeBit2 := FALSE;
   STATUS[432].EXT.ModeBit3 := FALSE;
   STATUS[432].EXT.BIT19 := FALSE;
   STATUS[432].EXT.BIT20 := FALSE;
   STATUS[432].EXT.AlarmSuppressed := FALSE;
   STATUS[432].EXT.AlarmPresent := FALSE;
   STATUS[432].EXT.AlarmFailUnAck := FALSE;
   STATUS[432].Status := 0;
   STATUS[432].TimeStamp := 16#0000;
   STATUS[433].EXT.AlarmWarnUnAck := FALSE;
   STATUS[433].EXT.AckRequired := FALSE;
   STATUS[433].EXT.Maintanence := FALSE;
   STATUS[433].EXT.Operation := FALSE;
   STATUS[433].EXT.Forced := FALSE;
   STATUS[433].EXT.BIT29 := FALSE;
   STATUS[433].EXT.BIT30 := FALSE;
   STATUS[433].EXT.BIT31 := FALSE;
   STATUS[433].EXT.ModeBit1 := FALSE;
   STATUS[433].EXT.ModeBit2 := FALSE;
   STATUS[433].EXT.ModeBit3 := FALSE;
   STATUS[433].EXT.BIT19 := FALSE;
   STATUS[433].EXT.BIT20 := FALSE;
   STATUS[433].EXT.AlarmSuppressed := FALSE;
   STATUS[433].EXT.AlarmPresent := FALSE;
   STATUS[433].EXT.AlarmFailUnAck := FALSE;
   STATUS[433].Status := 0;
   STATUS[433].TimeStamp := 16#0000;
   STATUS[434].EXT.AlarmWarnUnAck := FALSE;
   STATUS[434].EXT.AckRequired := FALSE;
   STATUS[434].EXT.Maintanence := FALSE;
   STATUS[434].EXT.Operation := FALSE;
   STATUS[434].EXT.Forced := FALSE;
   STATUS[434].EXT.BIT29 := FALSE;
   STATUS[434].EXT.BIT30 := FALSE;
   STATUS[434].EXT.BIT31 := FALSE;
   STATUS[434].EXT.ModeBit1 := FALSE;
   STATUS[434].EXT.ModeBit2 := FALSE;
   STATUS[434].EXT.ModeBit3 := FALSE;
   STATUS[434].EXT.BIT19 := FALSE;
   STATUS[434].EXT.BIT20 := FALSE;
   STATUS[434].EXT.AlarmSuppressed := FALSE;
   STATUS[434].EXT.AlarmPresent := FALSE;
   STATUS[434].EXT.AlarmFailUnAck := FALSE;
   STATUS[434].Status := 0;
   STATUS[434].TimeStamp := 16#0000;
   STATUS[435].EXT.AlarmWarnUnAck := FALSE;
   STATUS[435].EXT.AckRequired := FALSE;
   STATUS[435].EXT.Maintanence := FALSE;
   STATUS[435].EXT.Operation := FALSE;
   STATUS[435].EXT.Forced := FALSE;
   STATUS[435].EXT.BIT29 := FALSE;
   STATUS[435].EXT.BIT30 := FALSE;
   STATUS[435].EXT.BIT31 := FALSE;
   STATUS[435].EXT.ModeBit1 := FALSE;
   STATUS[435].EXT.ModeBit2 := FALSE;
   STATUS[435].EXT.ModeBit3 := FALSE;
   STATUS[435].EXT.BIT19 := FALSE;
   STATUS[435].EXT.BIT20 := FALSE;
   STATUS[435].EXT.AlarmSuppressed := FALSE;
   STATUS[435].EXT.AlarmPresent := FALSE;
   STATUS[435].EXT.AlarmFailUnAck := FALSE;
   STATUS[435].Status := 0;
   STATUS[435].TimeStamp := 16#0000;
   STATUS[436].EXT.AlarmWarnUnAck := FALSE;
   STATUS[436].EXT.AckRequired := FALSE;
   STATUS[436].EXT.Maintanence := FALSE;
   STATUS[436].EXT.Operation := FALSE;
   STATUS[436].EXT.Forced := FALSE;
   STATUS[436].EXT.BIT29 := FALSE;
   STATUS[436].EXT.BIT30 := FALSE;
   STATUS[436].EXT.BIT31 := FALSE;
   STATUS[436].EXT.ModeBit1 := FALSE;
   STATUS[436].EXT.ModeBit2 := FALSE;
   STATUS[436].EXT.ModeBit3 := FALSE;
   STATUS[436].EXT.BIT19 := FALSE;
   STATUS[436].EXT.BIT20 := FALSE;
   STATUS[436].EXT.AlarmSuppressed := FALSE;
   STATUS[436].EXT.AlarmPresent := FALSE;
   STATUS[436].EXT.AlarmFailUnAck := FALSE;
   STATUS[436].Status := 0;
   STATUS[436].TimeStamp := 16#0000;
   STATUS[437].EXT.AlarmWarnUnAck := FALSE;
   STATUS[437].EXT.AckRequired := FALSE;
   STATUS[437].EXT.Maintanence := FALSE;
   STATUS[437].EXT.Operation := FALSE;
   STATUS[437].EXT.Forced := FALSE;
   STATUS[437].EXT.BIT29 := FALSE;
   STATUS[437].EXT.BIT30 := FALSE;
   STATUS[437].EXT.BIT31 := FALSE;
   STATUS[437].EXT.ModeBit1 := FALSE;
   STATUS[437].EXT.ModeBit2 := FALSE;
   STATUS[437].EXT.ModeBit3 := FALSE;
   STATUS[437].EXT.BIT19 := FALSE;
   STATUS[437].EXT.BIT20 := FALSE;
   STATUS[437].EXT.AlarmSuppressed := FALSE;
   STATUS[437].EXT.AlarmPresent := FALSE;
   STATUS[437].EXT.AlarmFailUnAck := FALSE;
   STATUS[437].Status := 0;
   STATUS[437].TimeStamp := 16#0000;
   STATUS[438].EXT.AlarmWarnUnAck := FALSE;
   STATUS[438].EXT.AckRequired := FALSE;
   STATUS[438].EXT.Maintanence := FALSE;
   STATUS[438].EXT.Operation := FALSE;
   STATUS[438].EXT.Forced := FALSE;
   STATUS[438].EXT.BIT29 := FALSE;
   STATUS[438].EXT.BIT30 := FALSE;
   STATUS[438].EXT.BIT31 := FALSE;
   STATUS[438].EXT.ModeBit1 := FALSE;
   STATUS[438].EXT.ModeBit2 := FALSE;
   STATUS[438].EXT.ModeBit3 := FALSE;
   STATUS[438].EXT.BIT19 := FALSE;
   STATUS[438].EXT.BIT20 := FALSE;
   STATUS[438].EXT.AlarmSuppressed := FALSE;
   STATUS[438].EXT.AlarmPresent := FALSE;
   STATUS[438].EXT.AlarmFailUnAck := FALSE;
   STATUS[438].Status := 0;
   STATUS[438].TimeStamp := 16#0000;
   STATUS[439].EXT.AlarmWarnUnAck := FALSE;
   STATUS[439].EXT.AckRequired := FALSE;
   STATUS[439].EXT.Maintanence := FALSE;
   STATUS[439].EXT.Operation := FALSE;
   STATUS[439].EXT.Forced := FALSE;
   STATUS[439].EXT.BIT29 := FALSE;
   STATUS[439].EXT.BIT30 := FALSE;
   STATUS[439].EXT.BIT31 := FALSE;
   STATUS[439].EXT.ModeBit1 := FALSE;
   STATUS[439].EXT.ModeBit2 := FALSE;
   STATUS[439].EXT.ModeBit3 := FALSE;
   STATUS[439].EXT.BIT19 := FALSE;
   STATUS[439].EXT.BIT20 := FALSE;
